  1398 = 'Time / Hour Angle'
  991 = 'Time during which the pressure is built up'
  992 = 'Time during which the pressure is built up [s]'
  993 = 'Time needed for stopping the pumps [s]'
  1347 = 'Time processing status (by C++ task)'
  753 = 'Time to wait after electronics power off [s]'
  701 = 'Time to wait after electronics power on [s]'
  729 = 'Time to wait after move [s]'
  702 = 'Time to wait before powering off automatically [s]'
  1338 = 'Time to wait while powering off the pumps [s]'
  1337 = 'Time to wait while powering on the pumps  [s]'
  1339 = 'Time to wait while powering on the pumps [s]'
  1045 = 'Timeout for a fast movement [s]'
  1044 = 'Timeout for a movement [s]'
  57 = 'Timeout when closing [s]'
  56 = 'Timeout when opening [s]'
  796 = 'Timer\n4 sec'
  797 = 'Timer\nOFF\ndelay\n4 sec'
  477 = 'Timestamp update toggle (heartbeat)'
  363 = 'Timestamps'
  794 = 'TOF'
  795 = 'TOF\n4 sec'
  2013 = 'Tolerance (in degrees) for AZI to determine if it is at a known position'
  2014 = 'Tolerance (in degrees) for ELE to determine if it is at a known position'
  2015 = 'Tolerance (in degrees) for ROC to determine if it is at a known position'
  2016 = 'Tolerance (in degrees) for RON to determine if it is at a known position'
  62 = 'Tolerance at closed position [°]'
  60 = 'Tolerance at open position [°]'
  61 = 'Tolerance for standing still [°/s]'
  1781 = 'TOO LOW'
  33 = 'TOP'
  426 = 'Top'
  709 = 'top'
  778 = 'TOP 1'
  783 = 'Top 1'
  933 = 'Top 1 no underpressure'
  851 = 'Top 1 underpressure'
  878 = 'Top 1 underpressure OK'
  779 = 'TOP 2'
  784 = 'Top 2'
  935 = 'Top 2 no underpressure'
  852 = 'Top 2 underpressure'
  879 = 'Top 2 underpressure OK'
  780 = 'TOP 3'
  786 = 'Top 3'
  936 = 'Top 3 no underpressure'
  853 = 'Top 3 underpressure'
  880 = 'Top 3 underpressure OK'
  781 = 'TOP 4'
  787 = 'Top 4'
  937 = 'Top 4 no underpressure'
  854 = 'Top 4 underpressure'
  881 = 'Top 4 underpressure OK'
  961 = 'TOP drive'
  942 = 'Top no overpressure'
  785 = 'Top OP 3'
  855 = 'Top overpressure'
  886 = 'Top overpressure OK'
  984 = 'Top setpoint:'
  890 = 'Top TRIP OK'
  2096 = 'Torque'
  1542 = 'Torque command'
  1216 = 'Total time in milliseconds to repeat the pattern'
  2062 = "TPoint azimuth (' A' ) sign (-1 is negative, 1 is positive)"
  2066 = "TPoint azimuth (' A' ) sign correction (-1 is negative, 1 is positive)"
  2064 = 'TPoint delta azimuth sign correction (-1 is negative, 1 is positive)'
  2067 = 'TPoint delta elevation sign correction (-1 is negative, 1 is positive)'
  2063 = "TPoint elevation ('E' ) sign (-1 is negative, 1 is positive)"
  2065 = "TPoint elevation ('E' ) sign correction (-1 is negative, 1 is positive)"
  2059 = 'TPoint invert azimuth (A)'
  2061 = "TPoint invert azimuth (input ' A' )"
  2060 = 'TPoint invert azimuth (input A)'
  2068 = 'TPoint: use old formulas (different sign convention)'
  1437 = 'Track target after pointing'
  1774 = 'Track the new target after pointing'
  1775 = 'Track the target'
  1435 = 'Tracking'
  1760 = 'Transformations status (by C++ task)'
  73 = 'TRANSLATION'
  330 = 'Translation'
  142 = 'Translation position [mm]'
  141 = 'Translation position [°]'
  270 = 'Translation status'
  407 = 'Transmission status'
  1979 = 'travelled'
  1367 = 'Tropospheric lapse rate [K/m]'
  1414 = 'Troubleshoot'
  1418 = 'Troubleshoot \n& restart'
  1419 = 'Troubleshoot \nand restart'
  1417 = 'Troubleshoot & restart'
  1415 = 'Troubleshooting\n& restarting'
  1420 = 'Troubleshooting \nand restarting'
  1712 = 'True if a positive torque must be applied, false if a negative torque must be applied'
  1715 = 'True if the ABL torque must be applied in the same direction as the AZI acceleration'
  1716 = 'True if the AZI and ABL axes rotate in the same direction'
  1713 = 'True if the AZI and ABL axes rotate in the same direction, false if NOT'
  1714 = 'True if the AZI and ABL axes rotate in the same direction, false if not'
  2102 = 'True position'
  1826 = 'TRUE to invert the counting direction of the absolute encoder'
  1827 = 'TRUE to invert the counting direction of the LIDAs'
  1100 = 'Tube accelerometers'
  1465 = 'Tube flexure - sin(zeta) law'
  1467 = 'Tube flexure - tan(zeta) law'
  1281 = 'Turn off Cassegrain derotator'
  1279 = 'Turn off Nasmyth B derotator'
  1280 = 'Turn on Cassegrain derotator'
  1278 = 'Turn on Nasmyth B derotator'
  1029 = 'Turn on/off the circulation pump manually'
  1333 = 'Turn on/off the pumps manually'
  1466 = 'TX'
  296 = 'TxError counter:'
  1128 = 'Unblock'
  1133 = 'Unblock\n(Only staff can unblock from GUI)'
  1127 = 'Unblock\n(STAFF)'
  1134 = 'Unblock\n(Unblock from GUI = STAFF ONLY)'
  1135 = 'Unblock\n(Unblock from GUI = staff only)'
  1131 = 'Unblock\nforever'
  1132 = 'Unblock\nuntil re-initialize'
  1136 = 'Unblock \npermanently\n(until re-initialization)'
  1202 = 'Unblock button is being pushed'
  1137 = 'Unblock permanently\n(until re-initialization)'
  1140 = 'Unblock permanently\n(until safety is re-initialialized)'
  1141 = 'Unblock permanently\n(until Safety is re-initialized)'
  1126 = 'Unblock telescope'
  1139 = 'Unblocked permanently'
  817 = 'Under\npressure'
  772 = 'Underpressure'
  950 = 'Underpressure error'
  951 = 'Underpressure error detection'
  877 = 'Underpressure OK'
  777 = 'Underpressure status'
  776 = 'Underpressure summary'
  770 = 'Underpressure top 1'
  771 = 'Underpressure top 2'
  1442 = 'Units'
  413 = 'Unlock'
  1541 = 'UNLOCK'
  1805 = 'Unlock brake'
  1809 = 'Unlock brake temporarily'
  1535 = 'Update the (non-cyclic) values below'
  1534 = 'Update the non-cyclic values below'
  1505 = 'Update the values below'
  1331 = 'Use Cassegrain derotator'
  1332 = 'Use Nasmyth B derotator'
  1361 = 'Use relative humidity from sensors (not the value below)'
  1364 = 'Use relative humidity from telemetry (not the value below)'
  1358 = 'Use temperature from sensors (not the value below)'
  1363 = 'Use temperature from telemetry (not the value below)'
  1355 = 'Use temperatures from sensors (not from config)'
  1356 = 'Use temperatures from sensors (not the value below)'
  1610 = 'UT1'
  369 = 'UTC'
  372 = 'UTC date (y-m-s)'
  373 = 'UTC date (y-m-s) :'
  375 = 'UTC date (year-month-day) :'
  384 = 'UTC date (years - months - days)'
  381 = 'UTC date (years - months - days) :'
  380 = 'UTC date (years-months-days) :'
  374 = 'UTC date (yyyy-mm-dd) :'
  383 = 'UTC time (hours : minutes : seconds)'
  382 = 'UTC time (hours : minutes : seconds) :'
  376 = 'UTC time (hours:minutes:seconds) :'
  371 = 'UTC year/month/day'
  370 = 'UTC:'
  617 = 'Vacuum'
  618 = 'Vacuum OFF'
  643 = 'Vacuum ON'
  646 = 'Vacuum relay'
  173 = 'Value to write'
  120 = 'Vel. control Prop. term'
  122 = 'Vel. ctrl. Integral term'
  121 = 'Vel. ctrl. Proport. term'
  1738 = 'Velocities'
  1838 = 'Velocity'
  1683 = 'Velocity limit (bidirectional) of the physical axis in degrees/sec (>0)'
  1682 = 'Velocity limit (both directions) of the physical axis in degrees/sec (>0)'
  1679 = 'Velocity limit of the physical axis in degrees/sec (>0)'
  1720 = 'Velocity to search for the homing mark, in degrees/sec'
  1719 = 'Velocity when going to the start position, in degrees/sec'
  1292 = 'Verify fixed positions on thermal focus'
  836 = 'Verify if '
  837 = 'Verify if \nfrequency'
  838 = 'Verify if \nfrequency rises'
  839 = 'Verify if pumps\nfrequency rises'
  840 = 'Verify if pumps\nfrequency rises\n(QMin -> 0)'
  1463 = 'Vertical displacement of Nasmyth rotator'
  1621 = 'Virtual axis'
  1565 = 'W 270°'
  964 = 'Wait 2 minutes, so that the system can full start up in the background.'
  972 = 'Wait 2 minutes, so that the system can fully start up in the background.'
  1411 = 'Wake up'
  1427 = 'Wake up ...'
  1409 = 'Wake up telescope'
  1423 = 'Wake up the telescope'
  7 = 'WcState:'
  1657 = 'Which input (0-7) represents the negative limit switch?'
  1656 = 'Which input (0-7) represents the positive limit switch?'
  579 = 'with: RadialPressureSetpoint = CorrectionCoefficient * 1.33 bar * cos(elevation)'
  172 = 'Write'
  176 = 'Write config at initialization'
  688 = 'X'
  1106 = 'X angle'
  1285 = 'X fixed position tolerance [mm]'
  1284 = 'X fixed position [mm]'
  1 = 'XML config'
  150 = 'XML file'
  689 = 'Y'
  1287 = 'Y fixed position tolerance [mm]'
  1286 = 'Y fixed position [mm]'
  686 = 'Z'
  1077 = 'Z axis:'
  1255 = 'Z high speed'
  21 = '°'
  22 = '°/s'
  1758 = 'α'
  1856 = 'α offsetted'
  1854 = 'α travelled'
  1759 = 'δ'
  1858 = 'δ offsetted'
  1857 = 'δ travelled'
END_TEXTLIST

// ---- MTCS/Axes/Visu/VISU_AxesAzimuthAxis.TcVIS
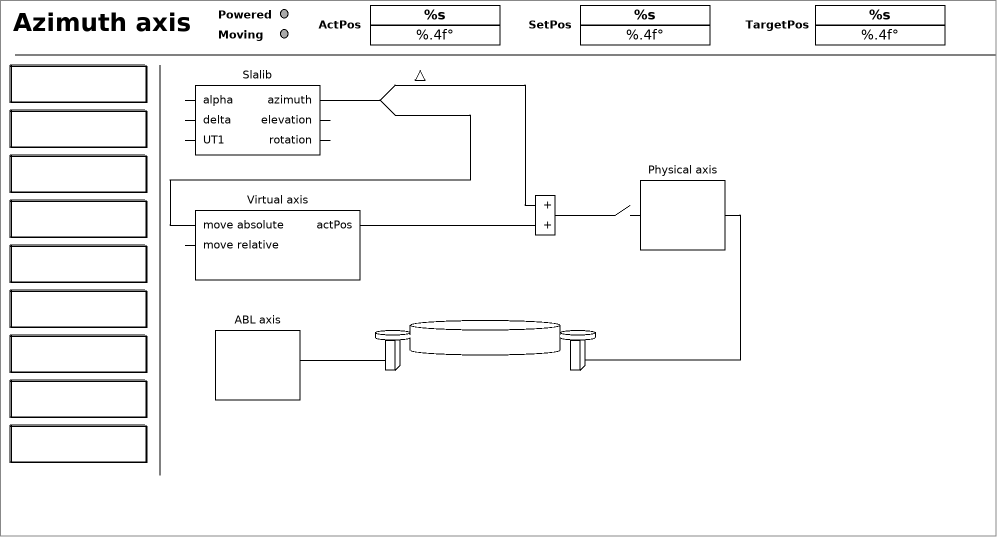
VISUALIZATION VISU_AxesAzimuthAxis  // 997x537
VAR_IN_OUT
	ref : AxesAzimuthAxis;
    ref_aziDriveChannel : AX52XXDriveChannel;
    ref_ablDriveChannel : AX52XXDriveChannel;
    widget : AxesAzimuthAxisWidget;
END_VAR
    Rectangle (10,0 195x45), "Azimuth axis"
    Frame (10,65 140x40)
        shows VISU_SubSubSystemButton(widget := widget.button_overview)
        OnMouseClick: FrameSelectionChange Selection=SelectedFrame=26eb0533-0645-4710-820d-78aa3cb40b18, GlobSel=AssignType=Directly, SelType=Locally
        OnMouseClick: execute { widget.activeTab := AxesAzimuthAxisTabs.OVERVIEW; }
    Frame (165,65 805x470)
        shows VISU_AxesAzimuthAxis_Overview(ref := ref, widget := widget)
        shows VISU_AxesAzimuthAxis_Processes(ref := ref, ref_aziDriveChannel := ref_aziDriveChannel, widget := widget)
        shows VISU_AX522DriveChannel(ref := ref_aziDriveChannel, widget := widget.aziDriveChannel)
        shows VISU_AX522DriveChannel(ref := ref_ablDriveChannel, widget := widget.ablDriveChannel)
        shows VISU_AngularAxis(axis := ref.parts.virtualAxis, widget := widget.virtualAxis)
        shows VISU_AngularAxis(axis := ref.parts.physicalAxis, widget := widget.physicalAxis)
        shows VISU_AngularAxis(axis := ref.parts.ablAxis, widget := widget.ablAxis)
        shows VISU_AxesAzimuthAxis_Lidas(ref := ref, widget := widget)
        shows VISU_AxesAzimuthAxis_AbsoluteEncoder(ref := ref, widget := widget)
        p4174417010: ref.parts.virtualAxis
        p2620823199: ref
    Line (160,475) (160,65)
    Frame (10,155 140x40)
        shows VISU_SubSubSystemButton(widget := widget.button_aziDriveChannel)
        OnMouseClick: FrameSelectionChange Selection=SelectedFrame=26eb0533-0645-4710-820d-78aa3cb40b18, Selection=2, GlobSel=AssignType=Directly, SelType=Locally
        OnMouseClick: execute { widget.activeTab := AxesAzimuthAxisTabs.AZI_DRIVE_CHANNEL; }
    Frame (10,200 140x40)
        shows VISU_SubSubSystemButton(widget := widget.button_ablDriveChannel)
        OnMouseClick: FrameSelectionChange Selection=SelectedFrame=26eb0533-0645-4710-820d-78aa3cb40b18, Selection=3, GlobSel=AssignType=Directly, SelType=Locally
        OnMouseClick: execute { widget.activeTab := AxesAzimuthAxisTabs.ABL_DRIVE_CHANNEL; }
    Frame (10,245 140x40)
        shows VISU_SubSubSystemButton(widget := widget.button_virtualAxis)
        OnMouseClick: FrameSelectionChange Selection=SelectedFrame=26eb0533-0645-4710-820d-78aa3cb40b18, Selection=4, GlobSel=AssignType=Directly, SelType=Locally
        OnMouseClick: execute { widget.activeTab := AxesAzimuthAxisTabs.VIRTUAL_AXIS; }
    Frame (10,290 140x40)
        shows VISU_SubSubSystemButton(widget := widget.button_physicalAxis)
        OnMouseClick: FrameSelectionChange Selection=SelectedFrame=26eb0533-0645-4710-820d-78aa3cb40b18, Selection=5, GlobSel=AssignType=Directly, SelType=Locally
        OnMouseClick: execute { widget.activeTab := AxesAzimuthAxisTabs.PHYSICAL_AXIS; }
    Frame (10,335 140x40)
        shows VISU_SubSubSystemButton(widget := widget.button_ablAxis)
        OnMouseClick: FrameSelectionChange Selection=SelectedFrame=26eb0533-0645-4710-820d-78aa3cb40b18, Selection=6, GlobSel=AssignType=Directly, SelType=Locally
        OnMouseClick: execute { widget.activeTab := AxesAzimuthAxisTabs.ABL_AXIS; }
    Frame (10,380 140x40)
        shows VISU_SubSubSystemButton(widget := widget.button_lidas)
        OnMouseClick: FrameSelectionChange Selection=SelectedFrame=26eb0533-0645-4710-820d-78aa3cb40b18, Selection=7, GlobSel=AssignType=Directly, SelType=Locally
        OnMouseClick: execute { widget.activeTab := AxesAzimuthAxisTabs.LIDAS; }
    Frame (10,425 140x40)
        shows VISU_SubSubSystemButton(widget := widget.button_absoluteEncoder)
        OnMouseClick: FrameSelectionChange Selection=SelectedFrame=26eb0533-0645-4710-820d-78aa3cb40b18, Selection=8, GlobSel=AssignType=Directly, SelType=Locally
        OnMouseClick: execute { widget.activeTab := AxesAzimuthAxisTabs.ABSOLUTE_ENCODER; }
    Frame (10,110 140x40)
        shows VISU_SubSubSystemButton(widget := widget.button_processes)
        OnMouseClick: FrameSelectionChange Selection=SelectedFrame=26eb0533-0645-4710-820d-78aa3cb40b18, Selection=1, GlobSel=AssignType=Directly, SelType=Locally
        OnMouseClick: execute { widget.activeTab := AxesAzimuthAxisTabs.PROCESSES; }
    Line (995,55) (15,55)
    Label (310,0 60x50), "ActPos"
    Rectangle (370,5 130x20), "%s", text variable: widget.actPos.dmsString
    Rectangle (370,25 130x20), "%.4f°", text variable: ref.actPos.degrees.value
    Label (520,0 60x50), "SetPos"
    Rectangle (580,5 130x20), "%s", text variable: widget.setPos.dmsString
    Rectangle (580,25 130x20), "%.4f°", text variable: ref.setPos.degrees.value
    Label (740,0 75x50), "TargetPos"
    Rectangle (815,5 130x20), "%s", text variable: widget.targetPos.dmsString
    Rectangle (815,25 130x20), "%.4f°", text variable: ref.targetPos.degrees.value
    Label (215,5 65x20), "Powered"
    Frame (280,5 10x15)
        shows VISU_State_gray_green(state := ref.statuses.poweredStatus.enabled)
    Label (215,25 65x20), "Moving"
    Frame (280,25 10x15)
        shows VISU_State_gray_green(state := ref.parts.physicalAxis.axis_ref.Status.Moving)
END_VISUALIZATION

// ---- MTCS/Axes/Visu/VISU_AxesAzimuthAxis_AbsoluteEncoder.TcVIS
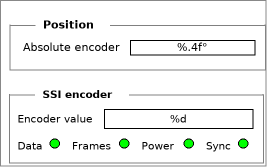
VISUALIZATION VISU_AxesAzimuthAxis_AbsoluteEncoder  // 267x167
VAR_IN_OUT
	ref : AxesAzimuthAxis;
    widget : AxesAzimuthAxisWidget;
END_VAR
    Frame (-5,80 270x85)
        shows VISU_SSIEncoder(ref := ref.parts.absoluteEncoder)
    Label (40,15 65x20), "Position"
    Polyline (110,25) (265,25) (265,70) (10,70) (10,25) (35,25)
    Label (20,40 105x15), "Absolute encoder"
    Rectangle (130,40 125x15), "%.4f°", text variable: ref.absoluteEncoderPosition.degrees.value
END_VISUALIZATION

// ---- MTCS/Axes/Visu/VISU_AxesAzimuthAxis_Processes.TcVIS
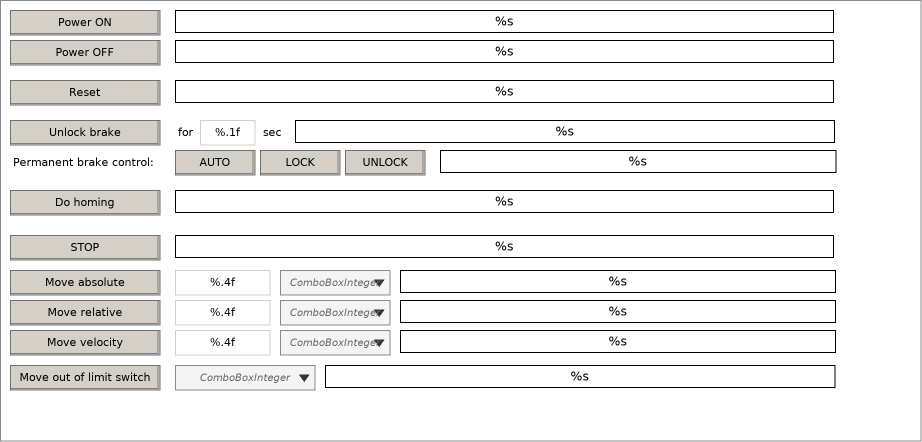
VISUALIZATION VISU_AxesAzimuthAxis_Processes  // 922x442
VAR_IN_OUT
	ref : AxesAzimuthAxis;
    ref_aziDriveChannel : AX52XXDriveChannel;
    widget : AxesAzimuthAxisWidget;
END_VAR
    Frame (10,10 910x55)
        shows VISU_Axes_Commands_Power(powerOn := ref.processes.powerOn, powerOff := ref.processes.powerOff, powerOnStatus := widget.processes_powerOnStatus, powerOffStatus := widget.processes_powerOffStatus)
    Frame (10,80 910x25)
        shows VISU_Axes_Commands_Reset(reset := ref.processes.reset, resetStatus := widget.processes_resetStatus)
    Frame (10,120 910x55)
        shows VISU_Axes_Commands_Brake(unlockBrake := ref.processes.unlockBrake, setBrake := ref_aziDriveChannel.processes.setBrake, unlockBrakeStatus := widget.processes_unlockBrakeStatus, setBrakeStatus := widget.aziDriveChannel.processes_setBrakeStatus)
    Frame (10,190 910x35)
        shows VISU_Axes_Commands_DoHoming(doHoming := ref.processes.doHoming, doHomingStatus := widget.processes_doHomingStatus)
    Frame (10,235 910x205)
        shows VISU_Axes_Commands_Movement(stop := ref.processes.stop, moveOutOfLimitSwitch := ref.processes.moveOutOfLimitSwitch, moveAbsolute := ref.processes.moveAbsolute, moveRelative := ref.processes.moveRelative, moveVelocity := ref.processes.moveVelocity, stopStatus := widget.processes_stopStatus, moveOutOfLimitSwitchStatus := widget.processes_moveOutOfLimitSwitchStatus, moveAbsoluteStatus := widget.processes_moveAbsoluteStatus, moveRelativeStatus := widget.processes_moveRelativeStatus, moveVelocityStatus := widget.processes_moveVelocityStatus)
END_VISUALIZATION

// ---- MTCS/Axes/Visu/VISU_AxesConfig_KnownPosition.TcVIS
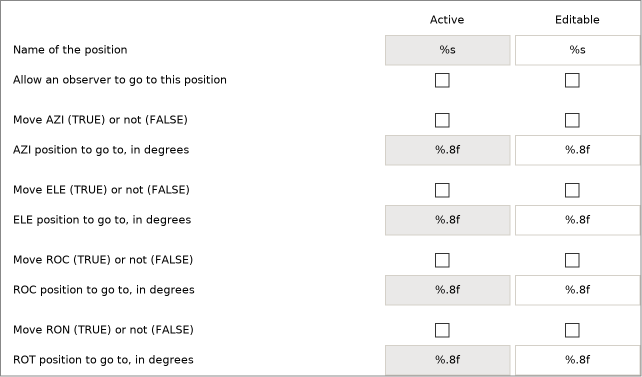
VISUALIZATION VISU_AxesConfig_KnownPosition  // 642x377
VAR_IN_OUT
    editable : AxesKnownPositionConfig;
	active : AxesKnownPositionConfig;
END_VAR
    Frame (385,35 255x30)
        shows VISU_ConfigStringEntry(active := active.name, editable := editable.name)
    Label (385,10 125x20), "Active"
    Label (515,10 125x20), "Editable"
    Label (10,35 370x30), "Name of the position"
    Frame (385,65 255x30)
        shows VISU_ConfigBOOLEntry(active := active.allowObserver, editable := editable.allowObserver)
    Label (10,65 370x30), "Allow an observer to go to this position"
    Label (10,135 370x30), "AZI position to go to, in degrees"
    Frame (385,135 255x30)
        shows VISU_ConfigLREAL8Entry(active := active.azi, editable := editable.azi)
    Label (10,105 370x30), "Move AZI (TRUE) or not (FALSE)"
    Frame (385,105 255x30)
        shows VISU_ConfigBOOLEntry(active := active.doAzi, editable := editable.doAzi)
    Label (10,205 370x30), "ELE position to go to, in degrees"
    Frame (385,205 255x30)
        shows VISU_ConfigLREAL8Entry(active := active.ele, editable := editable.ele)
    Label (10,175 370x30), "Move ELE (TRUE) or not (FALSE)"
    Frame (385,175 255x30)
        shows VISU_ConfigBOOLEntry(active := active.doEle, editable := editable.doEle)
    Label (10,275 370x30), "ROC position to go to, in degrees"
    Frame (385,275 255x30)
        shows VISU_ConfigLREAL8Entry(active := active.roc, editable := editable.roc)
    Label (10,245 370x30), "Move ROC (TRUE) or not (FALSE)"
    Frame (385,245 255x30)
        shows VISU_ConfigBOOLEntry(active := active.doRoc, editable := editable.doRoc)
    Label (10,345 370x30), "ROT position to go to, in degrees"
    Frame (385,345 255x30)
        shows VISU_ConfigLREAL8Entry(active := active.ron, editable := editable.ron)
    Label (10,315 370x30), "Move RON (TRUE) or not (FALSE)"
    Frame (385,315 255x30)
        shows VISU_ConfigBOOLEntry(active := active.doRon, editable := editable.doRon)
END_VISUALIZATION

// ---- MTCS/Axes/Visu/VISU_AxesConfig_KnownPositions.TcVIS
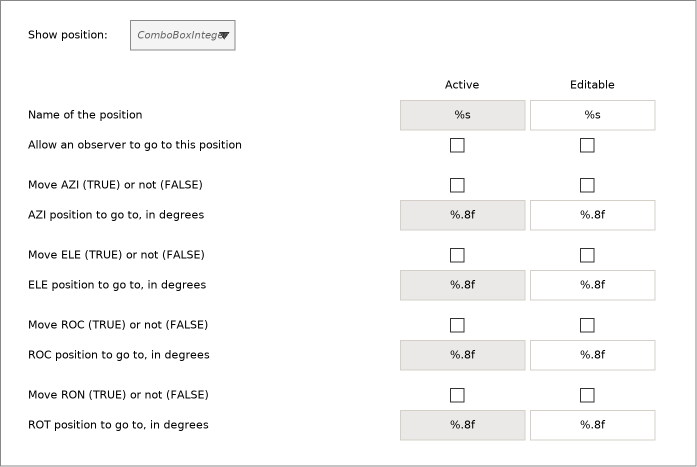
VISUALIZATION VISU_AxesConfig_KnownPositions  // 697x467
VAR_IN_OUT
    activePosition : INT;
    editable : AxesKnownPositionsConfig;
	active : AxesKnownPositionsConfig;
END_VAR
    Frame (15,65 680x400), frame switch variable: activePosition
        shows VISU_AxesConfig_KnownPosition(editable := editable.position0, active := active.position0)
        shows VISU_AxesConfig_KnownPosition(editable := editable.position1, active := active.position1)
        shows VISU_AxesConfig_KnownPosition(editable := editable.position2, active := active.position2)
        shows VISU_AxesConfig_KnownPosition(editable := editable.position3, active := active.position3)
        shows VISU_AxesConfig_KnownPosition(editable := editable.position4, active := active.position4)
        shows VISU_AxesConfig_KnownPosition(editable := editable.position5, active := active.position5)
        shows VISU_AxesConfig_KnownPosition(editable := editable.position6, active := active.position6)
        shows VISU_AxesConfig_KnownPosition(editable := editable.position7, active := active.position7)
        shows VISU_AxesConfig_KnownPosition(editable := editable.position8, active := active.position8)
        shows VISU_AxesConfig_KnownPosition(editable := editable.position9, active := active.position9)
        shows VISU_AxesConfig_KnownPosition(editable := editable.position10, active := active.position10)
        shows VISU_AxesConfig_KnownPosition(editable := editable.position11, active := active.position11)
        shows VISU_AxesConfig_KnownPosition(editable := editable.position12, active := active.position12)
        shows VISU_AxesConfig_KnownPosition(editable := editable.position13, active := active.position13)
        shows VISU_AxesConfig_KnownPosition(editable := editable.position14, active := active.position14)
        shows VISU_AxesConfig_KnownPosition(editable := editable.position15, active := active.position15)
        shows VISU_AxesConfig_KnownPosition(editable := editable.position16, active := active.position16)
        shows VISU_AxesConfig_KnownPosition(editable := editable.position17, active := active.position17)
        shows VISU_AxesConfig_KnownPosition(editable := editable.position18, active := active.position18)
        shows VISU_AxesConfig_KnownPosition(editable := editable.position19, active := active.position19)
    Label (25,20 150x30), "Show position:"
    ComboBoxInteger (130,20 105x30), variable: activePosition
END_VISUALIZATION

// ---- MTCS/Axes/Visu/VISU_AxesImage.TcVIS
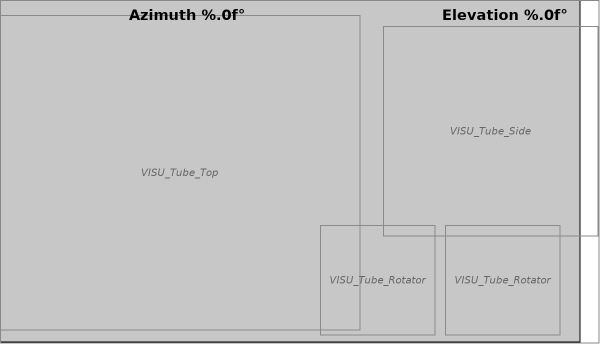
VISUALIZATION VISU_AxesImage  // 600x344
VAR_IN_OUT
	ref : Axes;
    widget : AxesWidget;
END_VAR
    Rectangle (0,0 580x342)
    Frame (383,26 215x210)
        shows VISU_Tube_Side(ele := widget.image.ele, eleTarget := widget.image.eleTarget, eleTargetInvisible := widget.image.eleTargetInvisible, mark10Degrees := widget.image.mark10Degrees)
    Frame (0,15 360x315)
        shows VISU_Tube_Top(widget := widget.image)
    Rectangle (90,5 195x20), "Azimuth %.0f°", text variable: ref.feedback.aziPos.degrees.value
    Rectangle (435,5 140x20), "Elevation %.0f°", text variable: ref.feedback.elePos.degrees.value
    Frame (320,225 115x110)
        shows VISU_Tube_Rotator(stationName := widget.image.rocStationName, name := widget.image.rocName, rotAngle := widget.image.roc)
    Frame (445,225 115x110)
        shows VISU_Tube_Rotator(stationName := widget.image.ronStationName, name := widget.image.ronName, rotAngle := widget.image.ron)
END_VISUALIZATION

// ---- MTCS/Axes/Visu/VISU_AxesManual_Offsets_AlphaDeltaRot.TcVIS
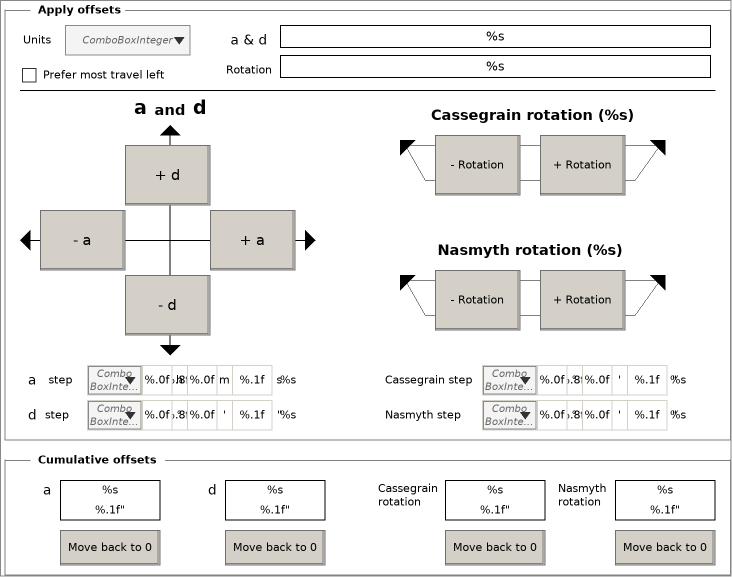
VISUALIZATION VISU_AxesManual_Offsets_AlphaDeltaRot  // 732x577
VAR_IN_OUT
	ref : Axes;
    widget : AxesManualOffsetsWidget;
END_VAR
    Polyline (165,460) (730,460) (730,575) (5,575) (5,460) (30,460)
    Polyline (125,10) (730,10) (730,440) (5,440) (5,10) (30,10)
    Polygon (660,145) (635,180) (425,180) (405,145)
    Line (170,350) (170,130)
    Line (25,240) (315,240)
    ComboBoxInteger (65,25 125x30), variable: widget.moveRelative.units, text list: 'AxesMoveAlphaDeltaProcessUnitsTextList'
    Rectangle (277,365 35x30), "%s", text variable: widget.pointRelative.unitsText, invisible if: widget.pointRelative.units = AxesMoveProcessWidgetUnits.DEGMINSEC
    Textfield (87,365 180x30), "%.8f", text variable: widget.pointRelative.field_alpha_decimal, invisible if: widget.pointRelative.units = AxesMoveProcessWidgetUnits.DEGMINSEC, input disabled if: widget.pointRelative.alphaDisabled
        OnMouseClick: write the text variable via VisuDialogs.Numpad
    Textfield (142,365 30x30), "%.0f", text variable: widget.pointRelative.field_alpha_h, invisible if: widget.pointRelative.units <> AxesMoveProcessWidgetUnits.DEGMINSEC, input disabled if: widget.pointRelative.alphaDisabled
        OnMouseClick: write the text variable via VisuDialogs.Numpad
    ComboBoxInteger (88,366 53x28), variable: widget.pointRelative.field_alpha_sign, invisible if: widget.pointRelative.units <> AxesMoveProcessWidgetUnits.DEGMINSEC, input disabled if: widget.pointRelative.alphaDisabled, text list: 'AxesDialogSignTextList'
    Textfield (187,365 30x30), "%.0f", text variable: widget.pointRelative.field_alpha_m, invisible if: widget.pointRelative.units <> AxesMoveProcessWidgetUnits.DEGMINSEC, input disabled if: widget.pointRelative.alphaDisabled
        OnMouseClick: write the text variable via VisuDialogs.Numpad
    Textfield (232,365 40x30), "%.1f", text variable: widget.pointRelative.field_alpha_s, invisible if: widget.pointRelative.units <> AxesMoveProcessWidgetUnits.DEGMINSEC, input disabled if: widget.pointRelative.alphaDisabled
        OnMouseClick: write the text variable via VisuDialogs.Numpad
    Label (172,365 15x30), "h", invisible if: widget.moveRelative.units <> AxesMoveProcessWidgetUnits.DEGMINSEC
    Label (217,365 15x30), "m", invisible if: widget.pointRelative.units <> AxesMoveProcessWidgetUnits.DEGMINSEC
    Label (272,365 15x30), "s", invisible if: widget.pointRelative.units <> AxesMoveProcessWidgetUnits.DEGMINSEC
    Rectangle (277,400 35x30), "%s", text variable: widget.pointRelative.unitsText, invisible if: widget.pointRelative.units = AxesMoveProcessWidgetUnits.DEGMINSEC
    Textfield (87,400 180x30), "%.8f", text variable: widget.pointRelative.field_delta_decimal, invisible if: widget.pointRelative.units = AxesMoveProcessWidgetUnits.DEGMINSEC, input disabled if: widget.pointRelative.deltaDisabled
        OnMouseClick: write the text variable via VisuDialogs.Numpad
    Textfield (142,400 30x30), "%.0f", text variable: widget.pointRelative.field_delta_d, invisible if: widget.pointRelative.units <> AxesMoveProcessWidgetUnits.DEGMINSEC, input disabled if: widget.pointRelative.deltaDisabled
        OnMouseClick: write the text variable via VisuDialogs.Numpad
    ComboBoxInteger (88,401 53x28), variable: widget.pointRelative.field_delta_sign, invisible if: widget.pointRelative.units <> AxesMoveProcessWidgetUnits.DEGMINSEC, input disabled if: widget.pointRelative.deltaDisabled, text list: 'AxesDialogSignTextList'
    Textfield (187,400 30x30), "%.0f", text variable: widget.pointRelative.field_delta_m, invisible if: widget.pointRelative.units <> AxesMoveProcessWidgetUnits.DEGMINSEC, input disabled if: widget.pointRelative.deltaDisabled
        OnMouseClick: write the text variable via VisuDialogs.Numpad
    Textfield (232,400 40x30), "%.1f", text variable: widget.pointRelative.field_delta_s, invisible if: widget.pointRelative.units <> AxesMoveProcessWidgetUnits.DEGMINSEC, input disabled if: widget.pointRelative.deltaDisabled
        OnMouseClick: write the text variable via VisuDialogs.Numpad
    Label (172,400 15x30), "°", invisible if: widget.moveRelative.units <> AxesMoveProcessWidgetUnits.DEGMINSEC
    Label (217,400 15x30), "'", invisible if: widget.moveRelative.units <> AxesMoveProcessWidgetUnits.DEGMINSEC
    Label (272,400 15x30), """, invisible if: widget.pointRelative.units <> AxesMoveProcessWidgetUnits.DEGMINSEC
    Rectangle (667,365 35x30), "%s", text variable: widget.moveRelative.unitsText, invisible if: widget.moveRelative.units = AxesMoveProcessWidgetUnits.DEGMINSEC
    Textfield (482,365 180x30), "%.8f", text variable: widget.moveRelative.field_roc_decimal, invisible if: widget.moveRelative.units = AxesMoveProcessWidgetUnits.DEGMINSEC, input disabled if: widget.moveRelative.rocDisabled
        OnMouseClick: write the text variable via VisuDialogs.Numpad
    Textfield (537,365 30x30), "%.0f", text variable: widget.moveRelative.field_roc_d, invisible if: widget.moveRelative.units <> AxesMoveProcessWidgetUnits.DEGMINSEC, input disabled if: widget.moveRelative.rocDisabled
        OnMouseClick: write the text variable via VisuDialogs.Numpad
    ComboBoxInteger (483,366 53x28), variable: widget.moveRelative.field_roc_sign, invisible if: widget.moveRelative.units <> AxesMoveProcessWidgetUnits.DEGMINSEC, input disabled if: widget.moveRelative.rocDisabled, text list: 'AxesDialogSignTextList'
    Textfield (582,365 30x30), "%.0f", text variable: widget.moveRelative.field_roc_m, invisible if: widget.moveRelative.units <> AxesMoveProcessWidgetUnits.DEGMINSEC, input disabled if: widget.moveRelative.rocDisabled
        OnMouseClick: write the text variable via VisuDialogs.Numpad
    Textfield (627,365 40x30), "%.1f", text variable: widget.moveRelative.field_roc_s, invisible if: widget.moveRelative.units <> AxesMoveProcessWidgetUnits.DEGMINSEC, input disabled if: widget.moveRelative.rocDisabled
        OnMouseClick: write the text variable via VisuDialogs.Numpad
    Label (567,365 15x30), "°", invisible if: widget.moveRelative.units <> AxesMoveProcessWidgetUnits.DEGMINSEC
    Label (612,365 15x30), "'", invisible if: widget.moveRelative.units <> AxesMoveProcessWidgetUnits.DEGMINSEC
    Label (667,365 15x30), """, invisible if: widget.moveRelative.units <> AxesMoveProcessWidgetUnits.DEGMINSEC
    Rectangle (667,400 35x30), "%s", text variable: widget.moveRelative.unitsText, invisible if: widget.moveRelative.units = AxesMoveProcessWidgetUnits.DEGMINSEC
    Textfield (482,400 180x30), "%.8f", text variable: widget.moveRelative.field_ron_decimal, invisible if: widget.moveRelative.units = AxesMoveProcessWidgetUnits.DEGMINSEC, input disabled if: widget.moveRelative.ronDisabled
        OnMouseClick: write the text variable via VisuDialogs.Numpad
    Textfield (537,400 30x30), "%.0f", text variable: widget.moveRelative.field_ron_d, invisible if: widget.moveRelative.units <> AxesMoveProcessWidgetUnits.DEGMINSEC, input disabled if: widget.moveRelative.ronDisabled
        OnMouseClick: write the text variable via VisuDialogs.Numpad
    ComboBoxInteger (483,401 53x28), variable: widget.moveRelative.field_ron_sign, invisible if: widget.moveRelative.units <> AxesMoveProcessWidgetUnits.DEGMINSEC, input disabled if: widget.moveRelative.ronDisabled, text list: 'AxesDialogSignTextList'
    Textfield (582,400 30x30), "%.0f", text variable: widget.moveRelative.field_ron_m, invisible if: widget.moveRelative.units <> AxesMoveProcessWidgetUnits.DEGMINSEC, input disabled if: widget.moveRelative.ronDisabled
        OnMouseClick: write the text variable via VisuDialogs.Numpad
    Textfield (627,400 40x30), "%.1f", text variable: widget.moveRelative.field_ron_s, invisible if: widget.moveRelative.units <> AxesMoveProcessWidgetUnits.DEGMINSEC, input disabled if: widget.moveRelative.ronDisabled
        OnMouseClick: write the text variable via VisuDialogs.Numpad
    Label (567,400 15x30), "°", invisible if: widget.moveRelative.units <> AxesMoveProcessWidgetUnits.DEGMINSEC
    Label (612,400 15x30), "'", invisible if: widget.moveRelative.units <> AxesMoveProcessWidgetUnits.DEGMINSEC
    Label (667,400 15x30), """, invisible if: widget.moveRelative.units <> AxesMoveProcessWidgetUnits.DEGMINSEC
    Frame (280,25 435x25)
        shows VISU_StatusWidget(widget := widget.pointRelative.actualStatus)
    Label (35,0 100x20), "Apply offsets"
    Button (125,145 85x60), "+ d", input disabled if: widget.pointRelative.deltaDisabled
        OnMouseClick: execute {
            ref.processes.pointRelative.request(
                alphaUnits := AxesAlphaUnits.DEGREES,
                alpha := 0.0,
                deltaunits := AxesDeltaUnits.DEGREES,
                delta := widget.pointRelative.deltaDeg);
        }
    Button (125,275 85x60), "- d", input disabled if: widget.pointRelative.deltaDisabled
        OnMouseClick: execute {
            ref.processes.pointRelative.request(
                alphaUnits := AxesAlphaUnits.DEGREES,
                alpha := 0.0,
                deltaunits := AxesDeltaUnits.DEGREES,
                delta := -widget.pointRelative.deltaDeg);
        }
    Button (210,210 85x60), "+ a", input disabled if: widget.pointRelative.alphaDisabled
        OnMouseClick: execute {
            ref.processes.pointRelative.request(
                alphaUnits := AxesAlphaUnits.DEGREES,
                alpha := widget.pointRelative.alphaDeg,
                deltaunits := AxesDeltaUnits.DEGREES,
                delta := 0.0);
        }
    Button (40,210 85x60), "- a", input disabled if: widget.pointRelative.alphaDisabled
        OnMouseClick: execute {
            ref.processes.pointRelative.request(
                alphaUnits := AxesAlphaUnits.DEGREES,
                alpha := -widget.pointRelative.alphaDeg,
                deltaunits := AxesDeltaUnits.DEGREES,
                delta := 0.0);
        }
    Label (42,365 35x30), "step"
    Label (42,400 40x30), "step"
    Button (540,135 85x60), "+ Rotation", input disabled if: widget.moveRelative.rocDisabled
        OnMouseClick: execute {
            ref.processes.moveRelative.request(
                units := AxesMoveUnits.DEGREES,
                azi := 0.0,
                ele := 0.0,
                rot := 0.0,
                roc := widget.moveRelative.rocDeg,
                ron := 0.0,
                doAzi := FALSE,
                doEle := FALSE,
                doRot := FALSE,
                doRoc := TRUE,
                doRon := FALSE,
                preferMostTravel := widget.preferMostTravel);
        }
    Button (435,135 85x60), "- Rotation", input disabled if: widget.moveRelative.rocDisabled
        OnMouseClick: execute {
            ref.processes.moveRelative.request(
                units := AxesMoveUnits.DEGREES,
                azi := 0.0,
                ele := 0.0,
                rot := 0.0,
                roc := -widget.moveRelative.rocDeg,
                ron := 0.0,
                doAzi := FALSE,
                doEle := FALSE,
                doRot := FALSE,
                doRoc := TRUE,
                doRon := FALSE,
                preferMostTravel := widget.preferMostTravel);
        }
    Polygon (160,135) (170,125) (180,135)
    Polygon (30,250) (20,240) (30,230)
    Polygon (305,250) (315,240) (305,230)
    Polygon (160,345) (170,355) (180,345)
    Polygon (665,155) (665,140) (650,140)
    Polygon (400,155) (415,140) (400,140)
    Label (382,365 100x30), "Cassegrain step"
    Label (382,400 100x30), "Nasmyth step"
    Label (20,25 55x30), "Units"
    Label (220,25 50x30), "a & d"
    Line (20,90) (715,90)
    Polygon (660,280) (635,315) (425,315) (405,280)
    Button (540,270 85x60), "+ Rotation", input disabled if: widget.moveRelative.ronDisabled
        OnMouseClick: execute {
            ref.processes.moveRelative.request(
                units := AxesMoveUnits.DEGREES,
                azi := 0.0,
                ele := 0.0,
                rot := 0.0,
                roc := 0.0,
                ron := widget.moveRelative.ronDeg,
                doAzi := FALSE,
                doEle := FALSE,
                doRot := FALSE,
                doRoc := FALSE,
                doRon := TRUE,
                preferMostTravel := widget.preferMostTravel);
        }
    Button (435,270 85x60), "- Rotation", input disabled if: widget.moveRelative.ronDisabled
        OnMouseClick: execute {
            ref.processes.moveRelative.request(
                units := AxesMoveUnits.DEGREES,
                azi := 0.0,
                ele := 0.0,
                rot := 0.0,
                roc := 0.0,
                ron := -widget.moveRelative.ronDeg,
                doAzi := FALSE,
                doEle := FALSE,
                doRot := FALSE,
                doRoc := FALSE,
                doRon := TRUE,
                preferMostTravel := widget.preferMostTravel);
        }
    Polygon (665,290) (665,275) (650,275)
    Polygon (400,290) (415,275) (400,275)
    Label (145,95 50x30), "and"
    Label (25,400 20x30), "d"
    Label (25,365 20x30), "a"
    Label (190,90 40x35), "d"
    Label (110,90 40x35), "a"
    Label (205,55 70x30), "Rotation"
    Frame (280,55 435x25)
        shows VISU_StatusWidget(widget := widget.moveRelative.actualStatus)
    Rectangle (60,480 100x20), "%s", text variable: widget.alphaOffsetted.hmsString
    Label (40,475 20x30), "a"
    Rectangle (60,500 100x20), "%.1f"", text variable: ref.target.alphaOffsetted.arcseconds.value
    Label (205,475 20x30), "d"
    Button (60,530 100x35), "Move back to 0", input disabled if: widget.pointRelative.alphaDisabled
        OnMouseClick: execute {
            ref.processes.pointRelative.request(
                alphaUnits := AxesAlphaUnits.DEGREES,
                alpha := -ref.target.alphaOffsetted.degrees.value,
                deltaunits := AxesDeltaUnits.DEGREES,
                delta := 0.0);
        }
    Label (35,450 120x20), "Cumulative offsets"
    Rectangle (60,480 100x40), colour toggle: widget.pointRelative.alphaDisabled
    Rectangle (225,480 100x20), "%s", text variable: widget.deltaOffsetted.dmsString
    Rectangle (225,500 100x20), "%.1f"", text variable: ref.target.deltaOffsetted.arcseconds.value
    Button (225,530 100x35), "Move back to 0", input disabled if: widget.pointRelative.deltaDisabled
        OnMouseClick: execute {
            ref.processes.pointRelative.request(
                alphaUnits := AxesAlphaUnits.DEGREES,
                alpha := 0.0,
                deltaunits := AxesDeltaUnits.DEGREES,
                delta := -ref.target.deltaOffsetted.degrees.value);
        }
    Rectangle (225,480 100x40), colour toggle: widget.pointRelative.deltaDisabled
    Rectangle (445,480 100x20), "%s", text variable: widget.rocTargetOffset.dmsString
    Rectangle (445,500 100x20), "%.1f"", text variable: ref.parts.roc.targetOffset.arcseconds.value
    Button (445,530 100x35), "Move back to 0", input disabled if: widget.moveRelative.rocDisabled
        OnMouseClick: execute {
            ref.processes.moveRelative.request(
                units := AxesMoveUnits.DEGREES,
                azi := 0.0,
                ele := 0.0,
                rot := 0.0,
                roc := -ref.parts.roc.targetOffset.degrees.value,
                ron := 0.0,
                doAzi := FALSE,
                doEle := FALSE,
                doRot := FALSE,
                doRoc := TRUE,
                doRon := FALSE, preferMostTravel := widget.preferMostTravel);
        }
    Rectangle (445,480 100x40), colour toggle: widget.moveRelative.rocDisabled
    Label (375,480 70x30), "Cassegrain rotation"
    Rectangle (615,480 100x20), "%s", text variable: widget.ronTargetOffset.dmsString
    Rectangle (615,500 100x20), "%.1f"", text variable: ref.parts.ron.targetOffset.arcseconds.value
    Button (615,530 100x35), "Move back to 0", input disabled if: widget.moveRelative.ronDisabled
        OnMouseClick: execute {
            ref.processes.moveRelative.request(
                units := AxesMoveUnits.DEGREES,
                azi := 0.0,
                ele := 0.0,
                rot := 0.0,
                roc := 0.0,
                ron :=  -ref.parts.ron.targetOffset.degrees.value,
                doAzi := FALSE,
                doEle := FALSE,
                doRot := FALSE,
                doRoc := FALSE,
                doRon := TRUE, preferMostTravel := widget.preferMostTravel);
        }
    Rectangle (615,480 100x40), colour toggle: widget.moveRelative.ronDisabled
    Label (555,480 60x30), "Nasmyth rotation"
    Rectangle (380,235 300x30), "Nasmyth rotation (%s)", text variable: ref.config.nasmythRotatorName
    Rectangle (380,100 305x30), "Cassegrain rotation (%s)", text variable: ref.config.cassegrainRotatorName
    Checkbox (20,60 195x30), "Prefer most travel left", variable: widget.preferMostTravel
END_VISUALIZATION

// ---- MTCS/Axes/Visu/VISU_AxesManual_Offsets_OLD.TcVIS
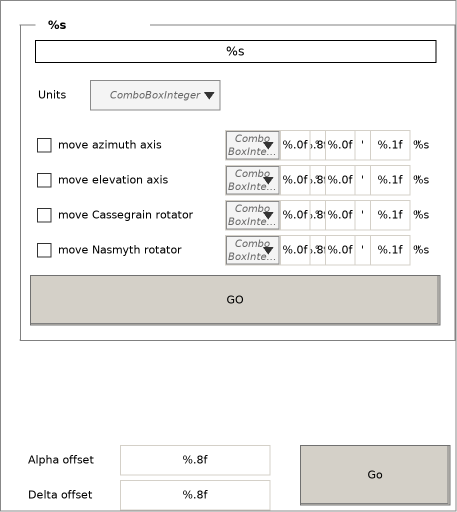
VISUALIZATION VISU_AxesManual_Offsets_OLD  // 457x512
VAR_IN_OUT
	ref : Axes;
    widget : AxesManualOffsetsWidget;
END_VAR
    Frame (15,10 440x370)
        shows VISU_AxesMultiMoveProcess(ref := ref.processes.moveRelative, widget := widget.moveRelative)
    Textfield (120,445 150x30), "%.8f", text variable: ref.processes.pointRelative.set.alpha
        OnMouseClick: write the text variable via VisuDialogs.Numpad
    Label (25,445 100x30), "Alpha offset"
    Textfield (120,480 150x30), "%.8f", text variable: ref.processes.pointRelative.set.delta
        OnMouseClick: write the text variable via VisuDialogs.Numpad
    Label (25,480 100x30), "Delta offset"
    Button (300,445 150x60), "Go", input disabled if: ref.processes.pointRelative.statuses.enabledStatus.disabled
        OnMouseClick: execute { ref.processes.pointRelative.do_request := TRUE; }
END_VISUALIZATION

// ---- MTCS/Axes/Visu/VISU_AxesRotationAxis_Processes.TcVIS
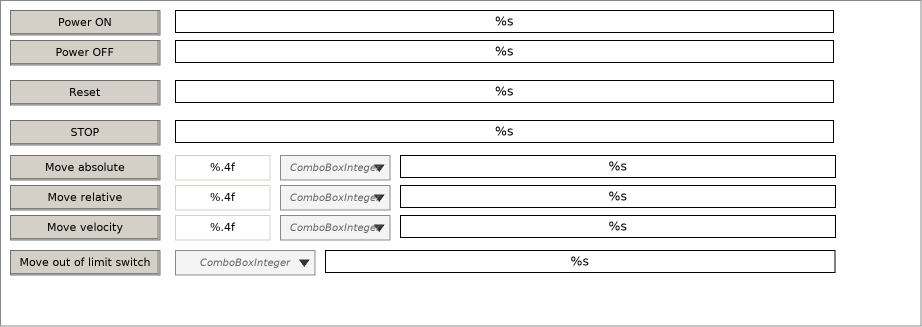
VISUALIZATION VISU_AxesRotationAxis_Processes  // 922x327
VAR_IN_OUT
	ref : AxesRotationAxis;
    ref_driveChannel : AX52XXDriveChannel;
    widget : AxesRotationAxisWidget;
END_VAR
    Frame (10,10 910x55)
        shows VISU_Axes_Commands_Power(powerOn := ref.processes.powerOn, powerOff := ref.processes.powerOff, powerOnStatus := widget.processes_powerOnStatus, powerOffStatus := widget.processes_powerOffStatus)
    Frame (10,80 910x25)
        shows VISU_Axes_Commands_Reset(reset := ref.processes.reset, resetStatus := widget.processes_resetStatus)
    Frame (10,120 910x205)
        shows VISU_Axes_Commands_Movement(stop := ref.processes.stop, moveOutOfLimitSwitch := ref.processes.moveOutOfLimitSwitch, moveAbsolute := ref.processes.moveAbsolute, moveRelative := ref.processes.moveRelative, moveVelocity := ref.processes.moveVelocity, stopStatus := widget.processes_stopStatus, moveOutOfLimitSwitchStatus := widget.processes_moveOutOfLimitSwitchStatus, moveAbsoluteStatus := widget.processes_moveAbsoluteStatus, moveRelativeStatus := widget.processes_moveRelativeStatus, moveVelocityStatus := widget.processes_moveVelocityStatus)
END_VISUALIZATION

// ---- MTCS/Axes/Visu/VISU_AxesRotationAxis_Overview.TcVIS
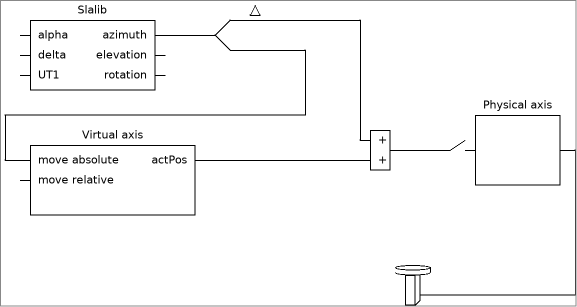
VISUALIZATION VISU_AxesRotationAxis_Overview  // 577x307
VAR_IN_OUT
	ref : AxesRotationAxis;
    widget : AxesRotationAxisWidget;
END_VAR
    Rectangle (405,275 10x30)
    Rectangle (30,20 125x70)
    Line (20,35) (30,35)
    Label (35,25 50x20), "alpha"
    Line (20,55) (30,55)
    Label (35,45 50x20), "delta"
    Line (20,75) (30,75)
    Label (35,65 50x20), "UT1"
    Polyline (255,5) (250,15) (260,15) (255,5)
    Label (30,0 125x20), "Slalib"
    Label (95,25 55x20), "azimuth"
    Label (90,45 60x20), "elevation"
    Label (100,65 50x20), "rotation"
    Line (155,55) (165,55)
    Line (155,75) (165,75)
    Rectangle (30,145 165x70)
    Label (35,150 95x20), "move absolute"
    Line (20,180) (30,180)
    Label (35,170 85x20), "move relative"
    Label (30,125 165x20), "Virtual axis"
    Label (135,150 55x20), "actPos"
    Polyline (155,35) (215,35) (230,50)
    Polyline (230,50) (305,50) (305,115) (5,115) (5,160) (30,160)
    Polyline (215,35) (230,20) (360,20) (360,140) (370,140)
    Polyline (195,160) (370,160)
    Rectangle (370,130 20x40)
    Label (375,130 15x20), "+"
    Label (375,150 15x20), "+"
    Line (390,150) (450,150)
    Line (450,150) (465,140)
    Line (465,150) (475,150)
    Rectangle (475,115 85x70)
    Label (475,95 85x20), "Physical axis"
    Polyline (560,150) (575,150) (575,295) (420,295)
    Polyline (415,305) (420,300) (420,275)
    Ellipse (395,270 35x5)
    Rectangle (395,270 35x2)
    Ellipse (395,265 35x5)
    Line (430,267) (430,272)
END_VISUALIZATION

// ---- MTCS/Axes/Visu/VISU_AxesElevationAxis_Processes.TcVIS
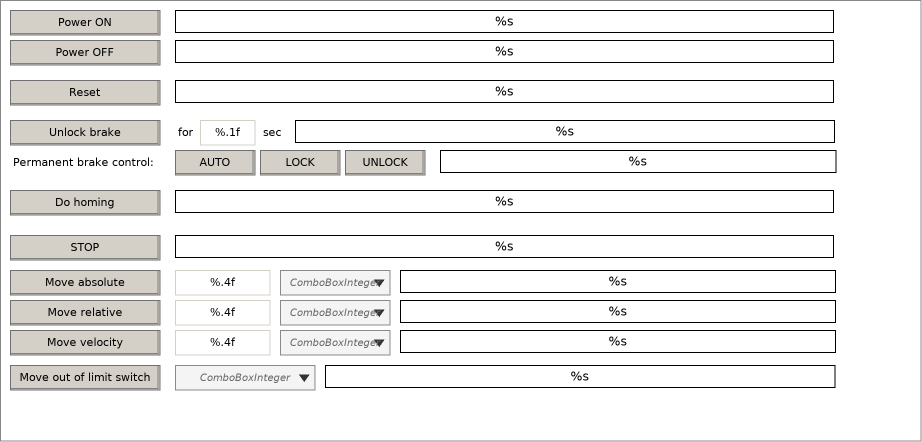
VISUALIZATION VISU_AxesElevationAxis_Processes  // 922x442
VAR_IN_OUT
	ref : AxesElevationAxis;
    ref_driveChannel : AX52XXDriveChannel;
    widget : AxesElevationAxisWidget;
END_VAR
    Frame (10,10 910x55)
        shows VISU_Axes_Commands_Power(powerOn := ref.processes.powerOn, powerOff := ref.processes.powerOff, powerOnStatus := widget.processes_powerOnStatus, powerOffStatus := widget.processes_powerOffStatus)
    Frame (10,80 910x25)
        shows VISU_Axes_Commands_Reset(reset := ref.processes.reset, resetStatus := widget.processes_resetStatus)
    Frame (10,120 910x55)
        shows VISU_Axes_Commands_Brake(unlockBrake := ref.processes.unlockBrake, setBrake := ref_driveChannel.processes.setBrake, unlockBrakeStatus := widget.processes_unlockBrakeStatus, setBrakeStatus := widget.driveChannel.processes_setBrakeStatus)
    Frame (10,190 910x35)
        shows VISU_Axes_Commands_DoHoming(doHoming := ref.processes.doHoming, doHomingStatus := widget.processes_doHomingStatus)
    Frame (10,235 910x205)
        shows VISU_Axes_Commands_Movement(stop := ref.processes.stop, moveOutOfLimitSwitch := ref.processes.moveOutOfLimitSwitch, moveAbsolute := ref.processes.moveAbsolute, moveRelative := ref.processes.moveRelative, moveVelocity := ref.processes.moveVelocity, stopStatus := widget.processes_stopStatus, moveOutOfLimitSwitchStatus := widget.processes_moveOutOfLimitSwitchStatus, moveAbsoluteStatus := widget.processes_moveAbsoluteStatus, moveRelativeStatus := widget.processes_moveRelativeStatus, moveVelocityStatus := widget.processes_moveVelocityStatus)
END_VISUALIZATION

// ---- MTCS/Axes/Visu/VISU_AxesManual_MoveVelocity.TcVIS
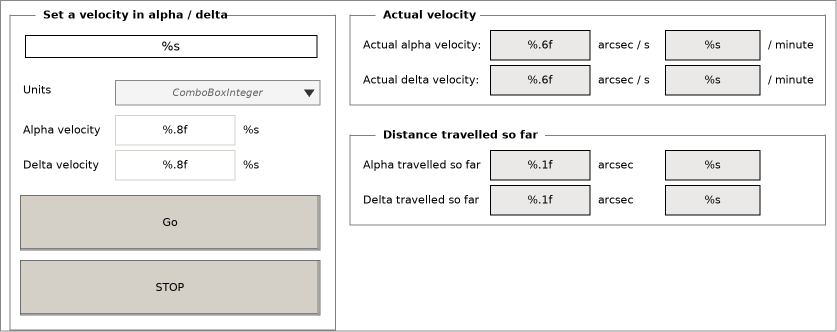
VISUALIZATION VISU_AxesManual_MoveVelocity  // 837x332
VAR_IN_OUT
	ref : Axes;
    widget : AxesManualMoveVelocityWidget;
END_VAR
    Polyline (225,15) (335,15) (335,330) (10,330) (10,15) (35,15)
    Polyline (480,15) (825,15) (825,105) (350,105) (350,15) (375,15)
    Label (380,5 100x20), "Actual velocity"
    Label (380,125 155x20), "Distance travelled so far"
    Polyline (545,135) (825,135) (825,225) (350,225) (350,135) (375,135)
    Textfield (115,115 120x30), "%.8f", text variable: widget.field_alphaVelocity
        OnMouseClick: write the text variable via VisuDialogs.Numpad
    Label (20,115 95x30), "Alpha velocity"
    Textfield (115,150 120x30), "%.8f", text variable: widget.field_deltaVelocity
        OnMouseClick: write the text variable via VisuDialogs.Numpad
    Label (20,150 95x30), "Delta velocity"
    Button (20,195 300x55), "Go", input disabled if: ref.processes.setAlphaDeltaVelocity.statuses.enabledStatus.disabled
        OnMouseClick: execute { widget.do_start := TRUE; }
    ComboBoxInteger (115,80 205x25), variable: widget.field_units, text list: 'AxesMoveVelocityUnitsTextList'
    Frame (25,35 295x25)
        shows VISU_StatusWidget(widget := widget.setAlphaDeltaVelocityStatus)
    Label (20,75 95x30), "Units"
    Rectangle (240,115 80x30), "%s", text variable: widget.label_units
    Label (360,30 145x30), "Actual alpha velocity:"
    Label (360,65 145x30), "Actual delta velocity:"
    Rectangle (490,30 100x30), "%.6f", text variable: ref.target.alphaVelocity.arcsecondsPerSecond.value
    Rectangle (490,65 100x30), "%.6f", text variable: ref.target.deltaVelocity.arcsecondsPerSecond.value
    Label (595,30 65x30), "arcsec / s"
    Rectangle (665,30 95x30), "%s", text variable: widget.alphaPerMinute.hmsString
    Rectangle (665,65 95x30), "%s", text variable: widget.deltaPerMinute.dmsString
    Label (765,30 70x30), "/ minute"
    Label (360,185 145x30), "Delta travelled so far"
    Label (360,150 145x30), "Alpha travelled so far"
    Rectangle (490,150 100x30), "%.1f", text variable: ref.target.alphaTravelled.arcseconds.value
    Rectangle (490,185 100x30), "%.1f", text variable: ref.target.deltaTravelled.arcseconds.value
    Label (595,150 75x30), "arcsec"
    Label (595,65 65x30), "arcsec / s"
    Label (765,65 70x30), "/ minute"
    Label (595,185 75x30), "arcsec"
    Rectangle (665,185 95x30), "%s", text variable: widget.deltaTravelledSoFar.dmsString
    Rectangle (665,150 95x30), "%s", text variable: widget.alphaTravelledSoFar.hmsString
    Button (20,260 300x55), "STOP", input disabled if: ref.processes.setAlphaDeltaVelocity.statuses.enabledStatus.disabled
        OnMouseClick: execute { widget.do_stop := TRUE; }
    Rectangle (240,150 80x30), "%s", text variable: widget.label_units
    Label (40,5 180x20), "Set a velocity in alpha / delta"
END_VISUALIZATION

// ---- MTCS/Axes/Visu/VISU_AxesManual_Offsets_AziEleRot.TcVIS
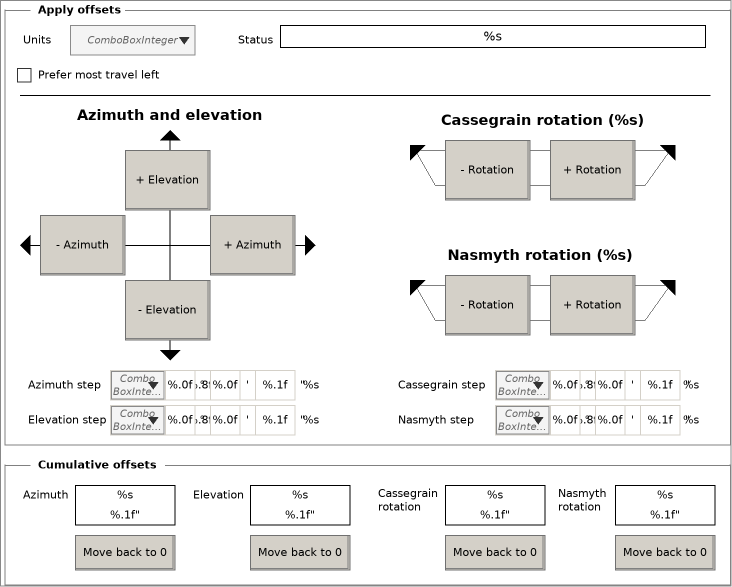
VISUALIZATION VISU_AxesManual_Offsets_AziEleRot  // 732x587
VAR_IN_OUT
	ref : Axes;
    widget : AxesManualOffsetsWidget;
END_VAR
    Polyline (125,10) (730,10) (730,445) (5,445) (5,10) (30,10)
    Polygon (670,150) (645,185) (435,185) (415,150)
    Line (170,355) (170,135)
    Line (25,245) (315,245)
    ComboBoxInteger (70,25 125x30), variable: widget.moveRelative.units, text list: 'AxesMoveProcessUnitsTextList'
    Rectangle (300,370 35x30), "%s", text variable: widget.moveRelative.unitsText, invisible if: widget.moveRelative.units = AxesMoveProcessWidgetUnits.DEGMINSEC
    Textfield (110,370 180x30), "%.8f", text variable: widget.moveRelative.field_azi_decimal, invisible if: widget.moveRelative.units = AxesMoveProcessWidgetUnits.DEGMINSEC, input disabled if: widget.moveRelative.aziDisabled
        OnMouseClick: write the text variable via VisuDialogs.Numpad
    Textfield (165,370 30x30), "%.0f", text variable: widget.moveRelative.field_azi_d, invisible if: widget.moveRelative.units <> AxesMoveProcessWidgetUnits.DEGMINSEC, input disabled if: widget.moveRelative.aziDisabled
        OnMouseClick: write the text variable via VisuDialogs.Numpad
    ComboBoxInteger (111,371 53x28), variable: widget.moveRelative.field_azi_sign, invisible if: widget.moveRelative.units <> AxesMoveProcessWidgetUnits.DEGMINSEC, input disabled if: widget.moveRelative.aziDisabled, text list: 'AxesDialogSignTextList'
    Textfield (210,370 30x30), "%.0f", text variable: widget.moveRelative.field_azi_m, invisible if: widget.moveRelative.units <> AxesMoveProcessWidgetUnits.DEGMINSEC, input disabled if: widget.moveRelative.aziDisabled
        OnMouseClick: write the text variable via VisuDialogs.Numpad
    Textfield (255,370 40x30), "%.1f", text variable: widget.moveRelative.field_azi_s, invisible if: widget.moveRelative.units <> AxesMoveProcessWidgetUnits.DEGMINSEC, input disabled if: widget.moveRelative.aziDisabled
        OnMouseClick: write the text variable via VisuDialogs.Numpad
    Label (195,370 15x30), "°", invisible if: widget.moveRelative.units <> AxesMoveProcessWidgetUnits.DEGMINSEC
    Label (240,370 15x30), "'", invisible if: widget.moveRelative.units <> AxesMoveProcessWidgetUnits.DEGMINSEC
    Label (295,370 15x30), """, invisible if: widget.moveRelative.units <> AxesMoveProcessWidgetUnits.DEGMINSEC
    Rectangle (300,405 35x30), "%s", text variable: widget.moveRelative.unitsText, invisible if: widget.moveRelative.units = AxesMoveProcessWidgetUnits.DEGMINSEC
    Textfield (110,405 180x30), "%.8f", text variable: widget.moveRelative.field_ele_decimal, invisible if: widget.moveRelative.units = AxesMoveProcessWidgetUnits.DEGMINSEC, input disabled if: widget.moveRelative.eleDisabled
        OnMouseClick: write the text variable via VisuDialogs.Numpad
    Textfield (165,405 30x30), "%.0f", text variable: widget.moveRelative.field_ele_d, invisible if: widget.moveRelative.units <> AxesMoveProcessWidgetUnits.DEGMINSEC, input disabled if: widget.moveRelative.eleDisabled
        OnMouseClick: write the text variable via VisuDialogs.Numpad
    ComboBoxInteger (111,406 53x28), variable: widget.moveRelative.field_ele_sign, invisible if: widget.moveRelative.units <> AxesMoveProcessWidgetUnits.DEGMINSEC, input disabled if: widget.moveRelative.eleDisabled, text list: 'AxesDialogSignTextList'
    Textfield (210,405 30x30), "%.0f", text variable: widget.moveRelative.field_ele_m, invisible if: widget.moveRelative.units <> AxesMoveProcessWidgetUnits.DEGMINSEC, input disabled if: widget.moveRelative.eleDisabled
        OnMouseClick: write the text variable via VisuDialogs.Numpad
    Textfield (255,405 40x30), "%.1f", text variable: widget.moveRelative.field_ele_s, invisible if: widget.moveRelative.units <> AxesMoveProcessWidgetUnits.DEGMINSEC, input disabled if: widget.moveRelative.eleDisabled
        OnMouseClick: write the text variable via VisuDialogs.Numpad
    Label (195,405 15x30), "°", invisible if: widget.moveRelative.units <> AxesMoveProcessWidgetUnits.DEGMINSEC
    Label (240,405 15x30), "'", invisible if: widget.moveRelative.units <> AxesMoveProcessWidgetUnits.DEGMINSEC
    Label (295,405 15x30), """, invisible if: widget.moveRelative.units <> AxesMoveProcessWidgetUnits.DEGMINSEC
    Rectangle (680,370 35x30), "%s", text variable: widget.moveRelative.unitsText, invisible if: widget.moveRelative.units = AxesMoveProcessWidgetUnits.DEGMINSEC
    Textfield (495,370 180x30), "%.8f", text variable: widget.moveRelative.field_roc_decimal, invisible if: widget.moveRelative.units = AxesMoveProcessWidgetUnits.DEGMINSEC, input disabled if: widget.moveRelative.rocDisabled
        OnMouseClick: write the text variable via VisuDialogs.Numpad
    Textfield (550,370 30x30), "%.0f", text variable: widget.moveRelative.field_roc_d, invisible if: widget.moveRelative.units <> AxesMoveProcessWidgetUnits.DEGMINSEC, input disabled if: widget.moveRelative.rocDisabled
        OnMouseClick: write the text variable via VisuDialogs.Numpad
    ComboBoxInteger (496,371 53x28), variable: widget.moveRelative.field_roc_sign, invisible if: widget.moveRelative.units <> AxesMoveProcessWidgetUnits.DEGMINSEC, input disabled if: widget.moveRelative.rocDisabled, text list: 'AxesDialogSignTextList'
    Textfield (595,370 30x30), "%.0f", text variable: widget.moveRelative.field_roc_m, invisible if: widget.moveRelative.units <> AxesMoveProcessWidgetUnits.DEGMINSEC, input disabled if: widget.moveRelative.rocDisabled
        OnMouseClick: write the text variable via VisuDialogs.Numpad
    Textfield (640,370 40x30), "%.1f", text variable: widget.moveRelative.field_roc_s, invisible if: widget.moveRelative.units <> AxesMoveProcessWidgetUnits.DEGMINSEC, input disabled if: widget.moveRelative.rocDisabled
        OnMouseClick: write the text variable via VisuDialogs.Numpad
    Label (580,370 15x30), "°", invisible if: widget.moveRelative.units <> AxesMoveProcessWidgetUnits.DEGMINSEC
    Label (625,370 15x30), "'", invisible if: widget.moveRelative.units <> AxesMoveProcessWidgetUnits.DEGMINSEC
    Label (680,370 15x30), """, invisible if: widget.moveRelative.units <> AxesMoveProcessWidgetUnits.DEGMINSEC
    Rectangle (680,405 35x30), "%s", text variable: widget.moveRelative.unitsText, invisible if: widget.moveRelative.units = AxesMoveProcessWidgetUnits.DEGMINSEC
    Textfield (495,405 180x30), "%.8f", text variable: widget.moveRelative.field_ron_decimal, invisible if: widget.moveRelative.units = AxesMoveProcessWidgetUnits.DEGMINSEC, input disabled if: widget.moveRelative.ronDisabled
        OnMouseClick: write the text variable via VisuDialogs.Numpad
    Textfield (550,405 30x30), "%.0f", text variable: widget.moveRelative.field_ron_d, invisible if: widget.moveRelative.units <> AxesMoveProcessWidgetUnits.DEGMINSEC, input disabled if: widget.moveRelative.ronDisabled
        OnMouseClick: write the text variable via VisuDialogs.Numpad
    ComboBoxInteger (496,406 53x28), variable: widget.moveRelative.field_ron_sign, invisible if: widget.moveRelative.units <> AxesMoveProcessWidgetUnits.DEGMINSEC, input disabled if: widget.moveRelative.ronDisabled, text list: 'AxesDialogSignTextList'
    Textfield (595,405 30x30), "%.0f", text variable: widget.moveRelative.field_ron_m, invisible if: widget.moveRelative.units <> AxesMoveProcessWidgetUnits.DEGMINSEC, input disabled if: widget.moveRelative.ronDisabled
        OnMouseClick: write the text variable via VisuDialogs.Numpad
    Textfield (640,405 40x30), "%.1f", text variable: widget.moveRelative.field_ron_s, invisible if: widget.moveRelative.units <> AxesMoveProcessWidgetUnits.DEGMINSEC, input disabled if: widget.moveRelative.ronDisabled
        OnMouseClick: write the text variable via VisuDialogs.Numpad
    Label (580,405 15x30), "°", invisible if: widget.moveRelative.units <> AxesMoveProcessWidgetUnits.DEGMINSEC
    Label (625,405 15x30), "'", invisible if: widget.moveRelative.units <> AxesMoveProcessWidgetUnits.DEGMINSEC
    Label (680,405 15x30), """, invisible if: widget.moveRelative.units <> AxesMoveProcessWidgetUnits.DEGMINSEC
    Frame (280,25 430x25)
        shows VISU_StatusWidget(widget := widget.moveRelative.actualStatus)
    Label (35,0 100x20), "Apply offsets"
    Button (125,150 85x60), "+ Elevation", input disabled if: widget.moveRelative.eleDisabled
        OnMouseClick: execute {
            ref.processes.moveRelative.request(
                units := AxesMoveUnits.DEGREES,
                azi := 0.0,
                ele := widget.moveRelative.eleDeg,
                rot := 0.0,
                roc := 0.0,
                ron := 0.0,
                doAzi := FALSE,
                doEle := TRUE,
                doRot := FALSE,
                doRoc := FALSE,
                doRon := FALSE,
                preferMostTravel := widget.preferMostTravel);
        }
    Button (125,280 85x60), "- Elevation", input disabled if: widget.moveRelative.eleDisabled
        OnMouseClick: execute {
            ref.processes.moveRelative.request(
                units := AxesMoveUnits.DEGREES,
                azi := 0.0,
                ele := -widget.moveRelative.eleDeg,
                rot := 0.0,
                roc := 0.0,
                ron := 0.0,
                doAzi := FALSE,
                doEle := TRUE,
                doRot := FALSE,
                doRoc := FALSE,
                doRon := FALSE,
                preferMostTravel := widget.preferMostTravel);
        }
    Button (210,215 85x60), "+ Azimuth", input disabled if: widget.moveRelative.aziDisabled
        OnMouseClick: execute {
            ref.processes.moveRelative.request(
                units := AxesMoveUnits.DEGREES,
                azi := widget.moveRelative.aziDeg,
                ele := 0.0,
                rot := 0.0,
                roc := 0.0,
                ron := 0.0,
                doAzi := TRUE,
                doEle := FALSE,
                doRot := FALSE,
                doRoc := FALSE,
                doRon := FALSE,
                preferMostTravel := widget.preferMostTravel);
        }
    Button (40,215 85x60), "- Azimuth", input disabled if: widget.moveRelative.aziDisabled
        OnMouseClick: execute {
            ref.processes.moveRelative.request(
                units := AxesMoveUnits.DEGREES,
                azi := -widget.moveRelative.aziDeg,
                ele := 0.0,
                rot := 0.0,
                roc := 0.0,
                ron := 0.0,
                doAzi := TRUE,
                doEle := FALSE,
                doRot := FALSE,
                doRoc := FALSE,
                doRon := FALSE,
                preferMostTravel := widget.preferMostTravel);
        }
    Label (25,370 80x30), "Azimuth step"
    Label (25,405 85x30), "Elevation step"
    Button (550,140 85x60), "+ Rotation", input disabled if: widget.moveRelative.rocDisabled
        OnMouseClick: execute {
            ref.processes.moveRelative.request(
                units := AxesMoveUnits.DEGREES,
                azi := 0.0,
                ele := 0.0,
                rot := 0.0,
                roc := widget.moveRelative.rocDeg,
                ron := 0.0,
                doAzi := FALSE,
                doEle := FALSE,
                doRot := FALSE,
                doRoc := TRUE,
                doRon := FALSE,
                preferMostTravel := widget.preferMostTravel);
        }
    Button (445,140 85x60), "- Rotation", input disabled if: widget.moveRelative.rocDisabled
        OnMouseClick: execute {
            ref.processes.moveRelative.request(
                units := AxesMoveUnits.DEGREES,
                azi := 0.0,
                ele := 0.0,
                rot := 0.0,
                roc := -widget.moveRelative.rocDeg,
                ron := 0.0,
                doAzi := FALSE,
                doEle := FALSE,
                doRot := FALSE,
                doRoc := TRUE,
                doRon := FALSE,
                preferMostTravel := widget.preferMostTravel);
        }
    Polygon (160,140) (170,130) (180,140)
    Polygon (30,255) (20,245) (30,235)
    Polygon (305,255) (315,245) (305,235)
    Polygon (160,350) (170,360) (180,350)
    Polygon (675,160) (675,145) (660,145)
    Polygon (410,160) (425,145) (410,145)
    Label (395,370 130x30), "Cassegrain step"
    Label (395,405 130x30), "Nasmyth step"
    Label (20,25 55x30), "Units"
    Label (235,25 45x30), "Status"
    Line (20,95) (710,95)
    Polygon (670,285) (645,320) (435,320) (415,285)
    Button (550,275 85x60), "+ Rotation", input disabled if: widget.moveRelative.ronDisabled
        OnMouseClick: execute {
            ref.processes.moveRelative.request(
                units := AxesMoveUnits.DEGREES,
                azi := 0.0,
                ele := 0.0,
                rot := 0.0,
                roc := 0.0,
                ron := widget.moveRelative.ronDeg,
                doAzi := FALSE,
                doEle := FALSE,
                doRot := FALSE,
                doRoc := FALSE,
                doRon := TRUE,
                preferMostTravel := widget.preferMostTravel);
        }
    Button (445,275 85x60), "- Rotation", input disabled if: widget.moveRelative.ronDisabled
        OnMouseClick: execute {
            ref.processes.moveRelative.request(
                units := AxesMoveUnits.DEGREES,
                azi := 0.0,
                ele := 0.0,
                rot := 0.0,
                roc := 0.0,
                ron := -widget.moveRelative.ronDeg,
                doAzi := FALSE,
                doEle := FALSE,
                doRot := FALSE,
                doRoc := FALSE,
                doRon := TRUE,
                preferMostTravel := widget.preferMostTravel);
        }
    Polygon (675,295) (675,280) (660,280)
    Polygon (410,295) (425,280) (410,280)
    Label (35,100 270x30), "Azimuth and elevation"
    Polyline (165,465) (730,465) (730,585) (5,585) (5,465) (30,465)
    Rectangle (75,485 100x20), "%s", text variable: widget.aziTargetOffset.dmsString
    Rectangle (75,505 100x20), "%.1f"", text variable: ref.parts.azi.targetOffset.arcseconds.value
    Button (75,535 100x35), "Move back to 0", input disabled if: widget.moveRelative.aziDisabled
        OnMouseClick: execute {
            ref.processes.moveRelative.request(
                units := AxesMoveUnits.DEGREES,
                azi := -ref.parts.azi.targetOffset.degrees.value,
                ele := 0.0,
                rot := 0.0,
                roc := 0.0,
                ron := 0.0,
                doAzi := TRUE,
                doEle := FALSE,
                doRot := FALSE,
                doRoc := FALSE,
                doRon := FALSE,
                preferMostTravel := widget.preferMostTravel);
        }
    Label (35,455 120x20), "Cumulative offsets"
    Rectangle (75,485 100x40), colour toggle: widget.moveRelative.aziDisabled
    Rectangle (250,485 100x20), "%s", text variable: widget.eleTargetOffset.dmsString
    Rectangle (250,505 100x20), "%.1f"", text variable: ref.parts.ele.targetOffset.arcseconds.value
    Button (250,535 100x35), "Move back to 0", input disabled if: widget.moveRelative.eleDisabled
        OnMouseClick: execute {
            ref.processes.moveRelative.request(
                units := AxesMoveUnits.DEGREES,
                azi := 0.0,
                ele := -ref.parts.ele.targetOffset.degrees.value,
                rot := 0.0,
                roc := 0.0,
                ron := 0.0,
                doAzi := FALSE,
                doEle := TRUE,
                doRot := FALSE,
                doRoc := FALSE,
                doRon := FALSE,
                preferMostTravel := widget.preferMostTravel);
        }
    Rectangle (250,485 100x40), colour toggle: widget.moveRelative.eleDisabled
    Rectangle (445,485 100x20), "%s", text variable: widget.rocTargetOffset.dmsString
    Rectangle (445,505 100x20), "%.1f"", text variable: ref.parts.roc.targetOffset.arcseconds.value
    Button (445,535 100x35), "Move back to 0", input disabled if: widget.moveRelative.rocDisabled
        OnMouseClick: execute {
            ref.processes.moveRelative.request(
                units := AxesMoveUnits.DEGREES,
                azi := 0.0,
                ele := 0.0,
                rot := 0.0,
                roc := -ref.parts.roc.targetOffset.degrees.value,
                ron := 0.0,
                doAzi := FALSE,
                doEle := FALSE,
                doRot := FALSE,
                doRoc := TRUE,
                doRon := FALSE,
                preferMostTravel := widget.preferMostTravel);
        }
    Rectangle (445,485 100x40), colour toggle: widget.moveRelative.rocDisabled
    Label (375,485 70x30), "Cassegrain rotation"
    Rectangle (615,485 100x20), "%s", text variable: widget.ronTargetOffset.dmsString
    Rectangle (615,505 100x20), "%.1f"", text variable: ref.parts.ron.targetOffset.arcseconds.value
    Button (615,535 100x35), "Move back to 0", input disabled if: widget.moveRelative.ronDisabled
        OnMouseClick: execute {
            ref.processes.moveRelative.request(
                units := AxesMoveUnits.DEGREES,
                azi := 0.0,
                ele := 0.0,
                rot := 0.0,
                roc := 0.0,
                ron :=  -ref.parts.ron.targetOffset.degrees.value,
                doAzi := FALSE,
                doEle := FALSE,
                doRot := FALSE,
                doRoc := FALSE,
                doRon := TRUE, preferMostTravel := widget.preferMostTravel);
        }
    Rectangle (615,485 100x40), colour toggle: widget.moveRelative.ronDisabled
    Label (555,485 60x30), "Nasmyth rotation"
    Label (20,485 55x20), "Azimuth"
    Label (190,485 55x20), "Elevation"
    Rectangle (390,240 300x30), "Nasmyth rotation (%s)", text variable: ref.config.nasmythRotatorName
    Rectangle (390,105 305x30), "Cassegrain rotation (%s)", text variable: ref.config.cassegrainRotatorName
    Checkbox (15,60 195x30), "Prefer most travel left", variable: widget.preferMostTravel
END_VISUALIZATION

// ---- MTCS/Axes/Visu/VISU_AxesManual_Joystick_AziEle.TcVIS
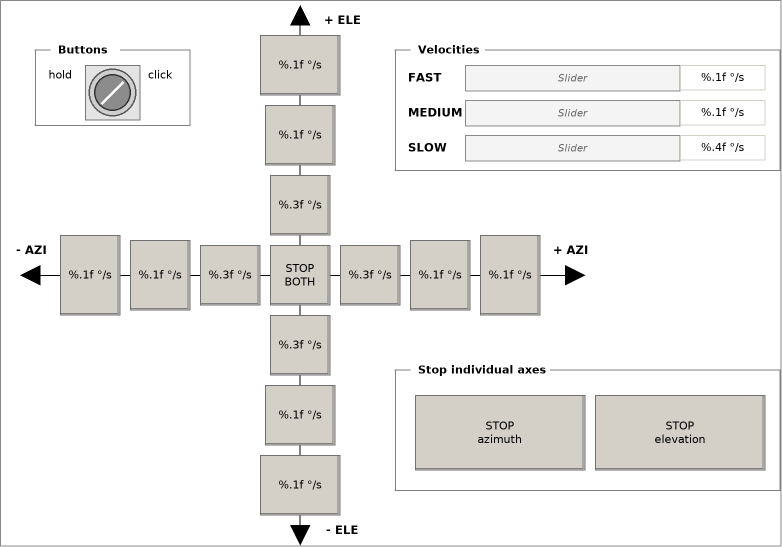
VISUALIZATION VISU_AxesManual_Joystick_AziEle  // 782x547
VAR_IN_OUT
	ref : Axes;
    widget : AxesManualJoystickAziEleWidget;
END_VAR
    Polyline (410,50) (395,50) (395,170) (780,170) (780,50) (485,50)
    Line (40,275) (575,275)
    Line (300,525) (300,25)
    Slider (465,65 215x26), variable: widget.joystick_velocity_fast, input disabled if: widget.joystick_disabled, scale 0..3
    Button (260,35 80x60), "%.1f °/s", text variable: widget.joystick_velocity_fast, input disabled if: widget.jog_ele_disabled
        tap widget.jog_ele_forward_fast
    Button (265,105 70x60), "%.1f °/s", text variable: widget.joystick_velocity_medium, input disabled if: widget.jog_ele_disabled
        tap widget.jog_ele_forward_medium
    Button (270,175 60x60), "%.3f °/s", text variable: widget.joystick_velocity_slow, input disabled if: widget.jog_ele_disabled
        tap widget.jog_ele_forward_slow
    Button (270,245 60x60), "STOP BOTH", input disabled if: ref.processes.stop.statuses.enabledStatus.disabled
        OnMouseClick: execute { ref.processes.stop.request(); }
    Button (260,455 80x60), "%.1f °/s", text variable: widget.joystick_velocity_fast, input disabled if: widget.jog_ele_disabled
        tap widget.jog_ele_backwards_fast
    Button (265,385 70x60), "%.1f °/s", text variable: widget.joystick_velocity_medium, input disabled if: widget.jog_ele_disabled
        tap widget.jog_ele_backwards_medium
    Button (270,315 60x60), "%.3f °/s", text variable: widget.joystick_velocity_slow, input disabled if: widget.jog_ele_disabled
        tap widget.jog_ele_backwards_slow
    Button (200,245 60x60), "%.3f °/s", text variable: widget.joystick_velocity_slow, input disabled if: widget.jog_azi_disabled
        tap widget.jog_azi_backwards_slow
    Button (130,240 60x70), "%.1f °/s", text variable: widget.joystick_velocity_medium, input disabled if: widget.jog_azi_disabled
        tap widget.jog_azi_backwards_medium
    Button (60,235 60x80), "%.1f °/s", text variable: widget.joystick_velocity_fast, input disabled if: widget.jog_azi_disabled
        tap widget.jog_azi_backwards_fast
    Button (480,235 60x80), "%.1f °/s", text variable: widget.joystick_velocity_fast, input disabled if: widget.jog_azi_disabled
        tap widget.jog_azi_forward_fast
    Button (410,240 60x70), "%.1f °/s", text variable: widget.joystick_velocity_medium, input disabled if: widget.jog_azi_disabled
        tap widget.jog_azi_forward_medium
    Button (340,245 60x60), "%.3f °/s", text variable: widget.joystick_velocity_slow, input disabled if: widget.jog_azi_disabled
        tap widget.jog_azi_forward_slow
    Textfield (680,65 85x25), "%.1f °/s", text variable: widget.joystick_velocity_fast, input disabled if: widget.joystick_disabled
        OnMouseClick: write the text variable via VisuDialogs.Numpad, min 0, max 3
    Polygon (290,25) (300,5) (310,25)
    Polygon (290,525) (300,545) (310,525)
    Polygon (565,285) (565,265) (585,275)
    Polygon (40,285) (40,265) (20,275)
    Label (405,65 70x25), "FAST"
    Slider (465,100 215x26), variable: widget.joystick_velocity_medium, input disabled if: widget.joystick_disabled, scale 0..3
    Label (405,100 70x25), "MEDIUM"
    Slider (465,135 215x26), variable: widget.joystick_velocity_slow, input disabled if: widget.joystick_disabled, scale 0..3
    Label (405,135 70x25), "SLOW"
    Label (415,40 70x20), "Velocities"
    Textfield (680,100 85x25), "%.1f °/s", text variable: widget.joystick_velocity_medium, input disabled if: widget.joystick_disabled
        OnMouseClick: write the text variable via VisuDialogs.Numpad, min 0, max 3
    Textfield (680,135 85x25), "%.4f °/s", text variable: widget.joystick_velocity_slow, input disabled if: widget.joystick_disabled
        OnMouseClick: write the text variable via VisuDialogs.Numpad, min 0, max 3
    Label (315,5 55x30), "+ ELE"
    Label (315,515 55x30), "- ELE"
    Label (550,235 45x30), "+ AZI"
    Label (10,235 40x30), "- AZI"
    Label (415,360 135x20), "Stop individual axes"
    Polyline (410,370) (395,370) (395,490) (780,490) (780,370) (550,370)
    Button (415,395 170x75), "STOP azimuth", input disabled if: ref.parts.azi.processes.stop.statuses.enabledStatus.disabled
        OnMouseClick: execute { ref.parts.azi.processes.stop.request(); }
    Button (595,395 170x75), "STOP elevation", input disabled if: ref.parts.ele.processes.stop.statuses.enabledStatus.disabled
        OnMouseClick: execute { ref.parts.ele.processes.stop.request(); }
    Polyline (50,50) (35,50) (35,125) (190,125) (190,50) (120,50)
    RotarySwitch (85,65 55x55), variable: widget.joystick_hold, input disabled if: widget.joystick_disabled, behaviour: TOGGLE, style: Switch-RotarySwitch-Gray
    Label (145,65 50x20), "click"
    Label (35,65 40x20), "hold"
    Label (55,40 65x20), "Buttons"
END_VISUALIZATION

// ---- MTCS/Axes/Visu/VISU_AxesManual_Joystick_Rot.TcVIS
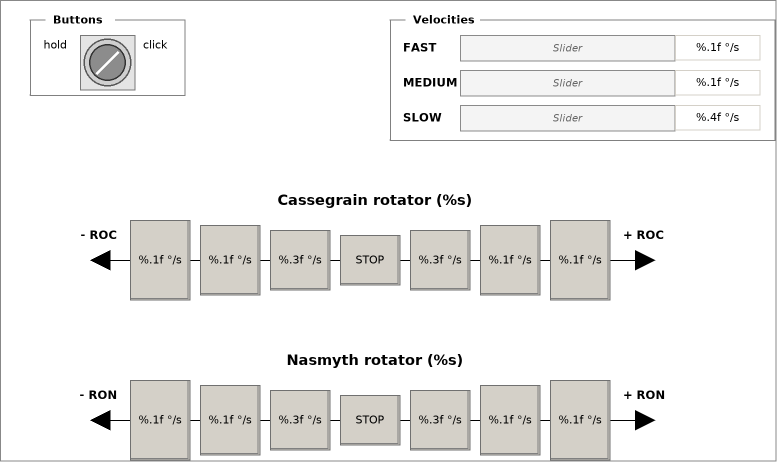
VISUALIZATION VISU_AxesManual_Joystick_Rot  // 777x462
VAR_IN_OUT
	ref : Axes;
    widget : AxesManualJoystickRotWidget;
END_VAR
    Polyline (405,20) (390,20) (390,140) (775,140) (775,20) (480,20)
    Line (110,260) (645,260)
    Slider (460,35 215x26), variable: widget.joystick_velocity_fast, input disabled if: widget.joystick_disabled, scale 0..3
    Button (270,230 60x60), "%.3f °/s", text variable: widget.joystick_velocity_slow, input disabled if: widget.jog_roc_disabled
        tap widget.jog_roc_backwards_slow
    Button (200,225 60x70), "%.1f °/s", text variable: widget.joystick_velocity_medium, input disabled if: widget.jog_roc_disabled
        tap widget.jog_roc_backwards_medium
    Button (130,220 60x80), "%.1f °/s", text variable: widget.joystick_velocity_fast, input disabled if: widget.jog_roc_disabled
        tap widget.jog_roc_backwards_fast
    Button (550,220 60x80), "%.1f °/s", text variable: widget.joystick_velocity_fast, input disabled if: widget.jog_roc_disabled
        tap widget.jog_roc_forward_fast
    Button (480,225 60x70), "%.1f °/s", text variable: widget.joystick_velocity_medium, input disabled if: widget.jog_roc_disabled
        tap widget.jog_roc_forward_medium
    Button (410,230 60x60), "%.3f °/s", text variable: widget.joystick_velocity_slow, input disabled if: widget.jog_roc_disabled
        tap widget.jog_roc_forward_slow
    Textfield (675,35 85x25), "%.1f °/s", text variable: widget.joystick_velocity_fast, input disabled if: widget.joystick_disabled
        OnMouseClick: write the text variable via VisuDialogs.Numpad, min 0, max 6
    Polygon (635,270) (635,250) (655,260)
    Polygon (110,270) (110,250) (90,260)
    Label (400,35 70x25), "FAST"
    Slider (460,70 215x26), variable: widget.joystick_velocity_medium, input disabled if: widget.joystick_disabled, scale 0..3
    Label (400,70 70x25), "MEDIUM"
    Slider (460,105 215x26), variable: widget.joystick_velocity_slow, input disabled if: widget.joystick_disabled, scale 0..3
    Label (400,105 70x25), "SLOW"
    Label (410,10 70x20), "Velocities"
    Textfield (675,70 85x25), "%.1f °/s", text variable: widget.joystick_velocity_medium, input disabled if: widget.joystick_disabled
        OnMouseClick: write the text variable via VisuDialogs.Numpad, min 0, max 3
    Textfield (675,105 85x25), "%.4f °/s", text variable: widget.joystick_velocity_slow, input disabled if: widget.joystick_disabled
        OnMouseClick: write the text variable via VisuDialogs.Numpad, min 0, max 3
    Label (620,220 45x30), "+ ROC"
    Label (80,220 40x30), "- ROC"
    Button (340,235 60x50), "STOP", input disabled if: widget.jog_roc_disabled
        OnMouseClick: execute { ref.parts.roc.processes.stop.request(); }
    Polyline (45,20) (30,20) (30,95) (185,95) (185,20) (115,20)
    RotarySwitch (80,35 55x55), variable: widget.joystick_hold, input disabled if: widget.joystick_disabled, behaviour: TOGGLE, style: Switch-RotarySwitch-Gray
    Label (140,35 50x20), "click"
    Label (30,35 40x20), "hold"
    Label (50,10 65x20), "Buttons"
    Line (110,420) (645,420)
    Button (270,390 60x60), "%.3f °/s", text variable: widget.joystick_velocity_slow, input disabled if: widget.jog_ron_disabled
        tap widget.jog_ron_backwards_slow
    Button (200,385 60x70), "%.1f °/s", text variable: widget.joystick_velocity_medium, input disabled if: widget.jog_ron_disabled
        tap widget.jog_ron_backwards_medium
    Button (130,380 60x80), "%.1f °/s", text variable: widget.joystick_velocity_fast, input disabled if: widget.jog_ron_disabled
        tap widget.jog_ron_backwards_fast
    Button (550,380 60x80), "%.1f °/s", text variable: widget.joystick_velocity_fast, input disabled if: widget.jog_ron_disabled
        tap widget.jog_ron_forward_fast
    Button (480,385 60x70), "%.1f °/s", text variable: widget.joystick_velocity_medium, input disabled if: widget.jog_ron_disabled
        tap widget.jog_ron_forward_medium
    Button (410,390 60x60), "%.3f °/s", text variable: widget.joystick_velocity_slow, input disabled if: widget.jog_ron_disabled
        tap widget.jog_ron_forward_slow
    Polygon (635,430) (635,410) (655,420)
    Polygon (110,430) (110,410) (90,420)
    Label (620,380 45x30), "+ RON"
    Label (80,380 40x30), "- RON"
    Button (340,395 60x50), "STOP", input disabled if: widget.jog_ron_disabled
        OnMouseClick: execute { ref.parts.ron.processes.stop.request(); }
    Rectangle (95,185 560x30), "Cassegrain rotator (%s)", text variable: ref.config.cassegrainRotatorName
    Rectangle (95,345 560x30), "Nasmyth rotator (%s)", text variable: ref.config.nasmythRotatorName
END_VISUALIZATION

// ---- MTCS/Axes/Visu/VISU_AxesManual_Positions.TcVIS
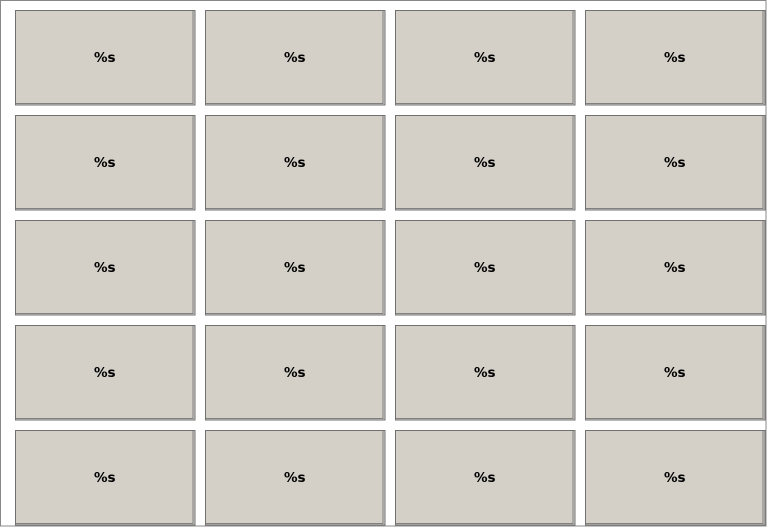
VISUALIZATION VISU_AxesManual_Positions  // 767x527
VAR_IN_OUT
	ref : Axes;
    widget : AxesManualPositionsWidget;
END_VAR
    Button (15,10 180x95), "%s", text variable: ref.config.knownPositions.position0.name, invisible if: widget.invisiblePosition0, input disabled if: ref.processes.moveKnownPosition.statuses.enabledStatus.disabled
        OnMouseClick: execute { ref.processes.moveKnownPosition.request(ref.config.knownPositions.position0.name); }
    Button (15,115 180x95), "%s", text variable: ref.config.knownPositions.position1.name, invisible if: widget.invisiblePosition1, input disabled if: ref.processes.moveKnownPosition.statuses.enabledStatus.disabled
        OnMouseClick: execute { ref.processes.moveKnownPosition.request(ref.config.knownPositions.position1.name); }
    Button (15,220 180x95), "%s", text variable: ref.config.knownPositions.position2.name, invisible if: widget.invisiblePosition2, input disabled if: ref.processes.moveKnownPosition.statuses.enabledStatus.disabled
        OnMouseClick: execute { ref.processes.moveKnownPosition.request(ref.config.knownPositions.position2.name); }
    Button (15,325 180x95), "%s", text variable: ref.config.knownPositions.position3.name, invisible if: widget.invisiblePosition3, input disabled if: ref.processes.moveKnownPosition.statuses.enabledStatus.disabled
        OnMouseClick: execute { ref.processes.moveKnownPosition.request(ref.config.knownPositions.position3.name); }
    Button (15,430 180x95), "%s", text variable: ref.config.knownPositions.position4.name, invisible if: widget.invisiblePosition4, input disabled if: ref.processes.moveKnownPosition.statuses.enabledStatus.disabled
        OnMouseClick: execute { ref.processes.moveKnownPosition.request(ref.config.knownPositions.position4.name); }
    Button (205,10 180x95), "%s", text variable: ref.config.knownPositions.position5.name, invisible if: widget.invisiblePosition5, input disabled if: ref.processes.moveKnownPosition.statuses.enabledStatus.disabled
        OnMouseClick: execute { ref.processes.moveKnownPosition.request(ref.config.knownPositions.position5.name); }
    Button (205,115 180x95), "%s", text variable: ref.config.knownPositions.position6.name, invisible if: widget.invisiblePosition6, input disabled if: ref.processes.moveKnownPosition.statuses.enabledStatus.disabled
        OnMouseClick: execute { ref.processes.moveKnownPosition.request(ref.config.knownPositions.position6.name); }
    Button (205,220 180x95), "%s", text variable: ref.config.knownPositions.position7.name, invisible if: widget.invisiblePosition7, input disabled if: ref.processes.moveKnownPosition.statuses.enabledStatus.disabled
        OnMouseClick: execute { ref.processes.moveKnownPosition.request(ref.config.knownPositions.position7.name); }
    Button (205,325 180x95), "%s", text variable: ref.config.knownPositions.position8.name, invisible if: widget.invisiblePosition8, input disabled if: ref.processes.moveKnownPosition.statuses.enabledStatus.disabled
        OnMouseClick: execute { ref.processes.moveKnownPosition.request(ref.config.knownPositions.position8.name); }
    Button (205,430 180x95), "%s", text variable: ref.config.knownPositions.position9.name, invisible if: widget.invisiblePosition9, input disabled if: ref.processes.moveKnownPosition.statuses.enabledStatus.disabled
        OnMouseClick: execute { ref.processes.moveKnownPosition.request(ref.config.knownPositions.position9.name); }
    Button (395,10 180x95), "%s", text variable: ref.config.knownPositions.position10.name, invisible if: widget.invisiblePosition10, input disabled if: ref.processes.moveKnownPosition.statuses.enabledStatus.disabled
        OnMouseClick: execute { ref.processes.moveKnownPosition.request(ref.config.knownPositions.position10.name); }
    Button (395,115 180x95), "%s", text variable: ref.config.knownPositions.position11.name, invisible if: widget.invisiblePosition11, input disabled if: ref.processes.moveKnownPosition.statuses.enabledStatus.disabled
        OnMouseClick: execute { ref.processes.moveKnownPosition.request(ref.config.knownPositions.position11.name); }
    Button (395,220 180x95), "%s", text variable: ref.config.knownPositions.position12.name, invisible if: widget.invisiblePosition12, input disabled if: ref.processes.moveKnownPosition.statuses.enabledStatus.disabled
        OnMouseClick: execute { ref.processes.moveKnownPosition.request(ref.config.knownPositions.position12.name); }
    Button (395,325 180x95), "%s", text variable: ref.config.knownPositions.position13.name, invisible if: widget.invisiblePosition13, input disabled if: ref.processes.moveKnownPosition.statuses.enabledStatus.disabled
        OnMouseClick: execute { ref.processes.moveKnownPosition.request(ref.config.knownPositions.position13.name); }
    Button (395,430 180x95), "%s", text variable: ref.config.knownPositions.position14.name, invisible if: widget.invisiblePosition14, input disabled if: ref.processes.moveKnownPosition.statuses.enabledStatus.disabled
        OnMouseClick: execute { ref.processes.moveKnownPosition.request(ref.config.knownPositions.position14.name); }
    Button (585,10 180x95), "%s", text variable: ref.config.knownPositions.position15.name, invisible if: widget.invisiblePosition15, input disabled if: ref.processes.moveKnownPosition.statuses.enabledStatus.disabled
        OnMouseClick: execute { ref.processes.moveKnownPosition.request(ref.config.knownPositions.position15.name); }
    Button (585,115 180x95), "%s", text variable: ref.config.knownPositions.position16.name, invisible if: widget.invisiblePosition16, input disabled if: ref.processes.moveKnownPosition.statuses.enabledStatus.disabled
        OnMouseClick: execute { ref.processes.moveKnownPosition.request(ref.config.knownPositions.position16.name); }
    Button (585,220 180x95), "%s", text variable: ref.config.knownPositions.position17.name, invisible if: widget.invisiblePosition17, input disabled if: ref.processes.moveKnownPosition.statuses.enabledStatus.disabled
        OnMouseClick: execute { ref.processes.moveKnownPosition.request(ref.config.knownPositions.position17.name); }
    Button (585,325 180x95), "%s", text variable: ref.config.knownPositions.position18.name, invisible if: widget.invisiblePosition18, input disabled if: ref.processes.moveKnownPosition.statuses.enabledStatus.disabled
        OnMouseClick: execute { ref.processes.moveKnownPosition.request(ref.config.knownPositions.position18.name); }
    Button (585,430 180x95), "%s", text variable: ref.config.knownPositions.position19.name, invisible if: widget.invisiblePosition19, input disabled if: ref.processes.moveKnownPosition.statuses.enabledStatus.disabled
        OnMouseClick: execute { ref.processes.moveKnownPosition.request(ref.config.knownPositions.position19.name); }
END_VISUALIZATION

// ---- MTCS/Axes/Visu/VISU_AxesManual_MoveAbsolute.TcVIS
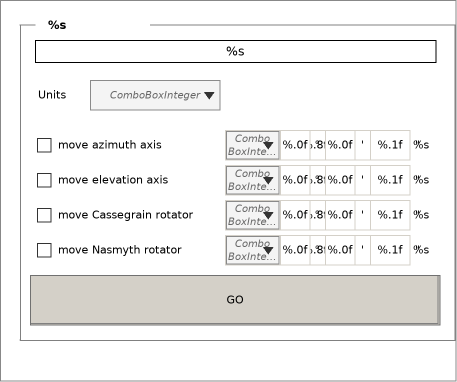
VISUALIZATION VISU_AxesManual_MoveAbsolute  // 457x382
VAR_IN_OUT
	ref : Axes;
    widget : AxesManualMoveAbsoluteWidget;
END_VAR
    Frame (15,10 440x370)
        shows VISU_AxesMultiMoveProcess(ref := ref.processes.moveAbsolute, widget := widget.moveAbsolute)
END_VISUALIZATION

// ---- MTCS/Axes/Visu/VISU_Axes_Commands_Power.TcVIS
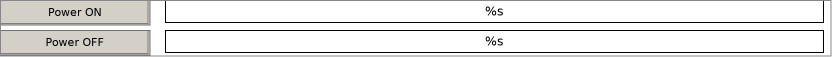
VISUALIZATION VISU_Axes_Commands_Power  // 832x57
VAR_IN_OUT
	powerOn : AxesPowerOnProcess;
    powerOff : AxesPowerOffProcess;
    
    powerOnStatus : StatusWidget;
    powerOffStatus : StatusWidget;
    
END_VAR
    Button (0,0 150x25), "Power ON", input disabled if: powerOn.statuses.enabledStatus.disabled
        OnMouseClick: execute { powerOn.request(); }
    Button (0,30 150x25), "Power OFF", input disabled if: powerOff.statuses.enabledStatus.disabled
        OnMouseClick: execute { powerOff.request(); }
    Frame (165,0 665x25)
        shows VISU_StatusWidget(widget := powerOnStatus)
    Frame (165,30 665x25)
        shows VISU_StatusWidget(widget := powerOffStatus)
END_VISUALIZATION

// ---- MTCS/Axes/Visu/VISU_AxesElevationAxis_Overview.TcVIS
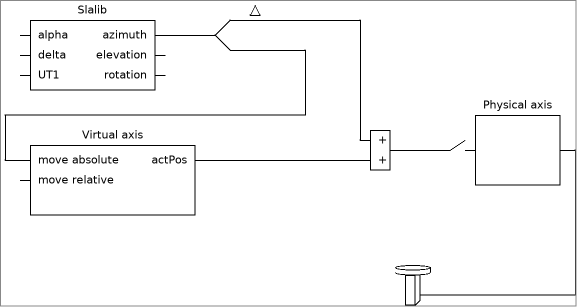
VISUALIZATION VISU_AxesElevationAxis_Overview  // 577x307
VAR_IN_OUT
	ref : AxesElevationAxis;
    widget : AxesElevationAxisWidget;
END_VAR
    Rectangle (405,275 10x30)
    Rectangle (30,20 125x70)
    Line (20,35) (30,35)
    Label (35,25 50x20), "alpha"
    Line (20,55) (30,55)
    Label (35,45 50x20), "delta"
    Line (20,75) (30,75)
    Label (35,65 50x20), "UT1"
    Polyline (255,5) (250,15) (260,15) (255,5)
    Label (30,0 125x20), "Slalib"
    Label (95,25 55x20), "azimuth"
    Label (90,45 60x20), "elevation"
    Label (100,65 50x20), "rotation"
    Line (155,55) (165,55)
    Line (155,75) (165,75)
    Rectangle (30,145 165x70)
    Label (35,150 95x20), "move absolute"
    Line (20,180) (30,180)
    Label (35,170 85x20), "move relative"
    Label (30,125 165x20), "Virtual axis"
    Label (135,150 55x20), "actPos"
    Polyline (155,35) (215,35) (230,50)
    Polyline (230,50) (305,50) (305,115) (5,115) (5,160) (30,160)
    Polyline (215,35) (230,20) (360,20) (360,140) (370,140)
    Polyline (195,160) (370,160)
    Rectangle (370,130 20x40)
    Label (375,130 15x20), "+"
    Label (375,150 15x20), "+"
    Line (390,150) (450,150)
    Line (450,150) (465,140)
    Line (465,150) (475,150)
    Rectangle (475,115 85x70)
    Label (475,95 85x20), "Physical axis"
    Polyline (560,150) (575,150) (575,295) (420,295)
    Polyline (415,305) (420,300) (420,275)
    Ellipse (395,270 35x5)
    Rectangle (395,270 35x2)
    Ellipse (395,265 35x5)
    Line (430,267) (430,272)
END_VISUALIZATION

// ---- MTCS/Axes/Visu/VISU_AxesElevationAxis_AbsoluteEncoder.TcVIS
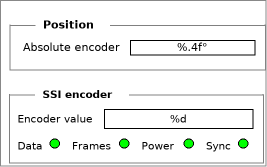
VISUALIZATION VISU_AxesElevationAxis_AbsoluteEncoder  // 267x167
VAR_IN_OUT
	ref : AxesElevationAxis;
    widget : AxesElevationAxisWidget;
END_VAR
    Frame (-5,80 270x85)
        shows VISU_SSIEncoder(ref := ref.parts.absoluteEncoder)
    Label (40,15 65x20), "Position"
    Polyline (110,25) (265,25) (265,70) (10,70) (10,25) (35,25)
    Label (20,40 105x15), "Absolute encoder"
    Rectangle (130,40 125x15), "%.4f°", text variable: ref.absoluteEncoderPosition.degrees.value
END_VISUALIZATION

// ---- MTCS/Axes/Visu/VISU_AxesElevationAxis_Lidas.TcVIS
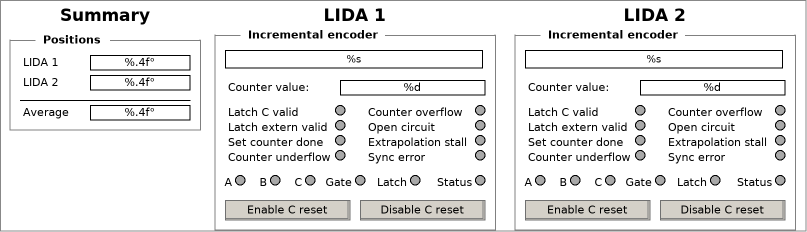
VISUALIZATION VISU_AxesElevationAxis_Lidas  // 807x232
VAR_IN_OUT
	ref : AxesElevationAxis;
    widget : AxesElevationAxisWidget;
END_VAR
    Label (215,0 280x30), "LIDA 1"
    Frame (215,25 290x205)
        shows VISU_IncrementalEncoder(ref := ref.parts.lida1, widget := widget.lida1)
    Label (515,0 280x30), "LIDA 2"
    Frame (515,25 290x205)
        shows VISU_IncrementalEncoder(ref := ref.parts.lida2, widget := widget.lida2)
    Label (10,0 190x30), "Summary"
    Label (40,30 65x20), "Positions"
    Polyline (110,40) (200,40) (200,130) (10,130) (10,40) (35,40)
    Label (20,55 90x15), "LIDA 1"
    Rectangle (90,55 100x15), "%.4f°", text variable: ref.lida1Position.degrees.value
    Rectangle (90,75 100x15), "%.4f°", text variable: ref.lida2Position.degrees.value
    Label (20,75 90x15), "LIDA 2"
    Label (20,105 90x15), "Average"
    Rectangle (90,105 100x15), "%.4f°", text variable: ref.lidaAveragePosition.degrees.value
    Line (20,100) (190,100)
END_VISUALIZATION

// ---- MTCS/Axes/Visu/VISU_AxesAzimuthAxis_Overview.TcVIS
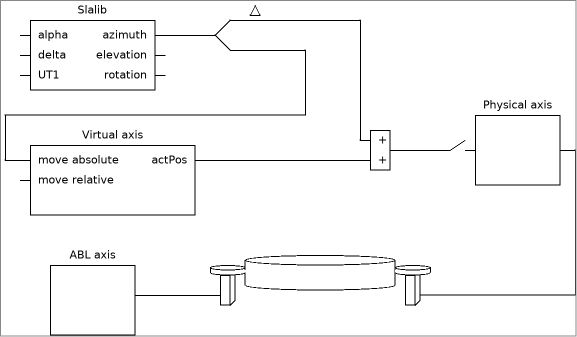
VISUALIZATION VISU_AxesAzimuthAxis_Overview  // 577x337
VAR_IN_OUT
	ref : AxesAzimuthAxis;
    widget : AxesAzimuthAxisWidget;
END_VAR
    Rectangle (405,275 10x30)
    Rectangle (30,20 125x70)
    Line (20,35) (30,35)
    Label (35,25 50x20), "alpha"
    Line (20,55) (30,55)
    Label (35,45 50x20), "delta"
    Line (20,75) (30,75)
    Label (35,65 50x20), "UT1"
    Polyline (255,5) (250,15) (260,15) (255,5)
    Label (30,0 125x20), "Slalib"
    Label (95,25 55x20), "azimuth"
    Label (90,45 60x20), "elevation"
    Label (100,65 50x20), "rotation"
    Line (155,55) (165,55)
    Line (155,75) (165,75)
    Rectangle (30,145 165x70)
    Label (35,150 95x20), "move absolute"
    Line (20,180) (30,180)
    Label (35,170 85x20), "move relative"
    Label (30,125 165x20), "Virtual axis"
    Label (135,150 55x20), "actPos"
    Polyline (155,35) (215,35) (230,50)
    Polyline (230,50) (305,50) (305,115) (5,115) (5,160) (30,160)
    Polyline (215,35) (230,20) (360,20) (360,140) (370,140)
    Polyline (195,160) (370,160)
    Rectangle (370,130 20x40)
    Label (375,130 15x20), "+"
    Label (375,150 15x20), "+"
    Line (390,150) (450,150)
    Line (450,150) (465,140)
    Line (465,150) (475,150)
    Rectangle (475,115 85x70)
    Label (475,95 85x20), "Physical axis"
    Polyline (560,150) (575,150) (575,295) (420,295)
    Rectangle (50,265 85x70)
    Label (50,245 85x20), "ABL axis"
    Ellipse (245,280 150x10)
    Rectangle (245,260 150x25)
    Ellipse (245,255 150x10)
    Line (245,285) (245,260)
    Line (395,285) (395,260)
    Polyline (415,305) (420,300) (420,275)
    Ellipse (395,270 35x5)
    Rectangle (395,270 35x2)
    Ellipse (395,265 35x5)
    Line (430,267) (430,272)
    Rectangle (220,275 10x30)
    Polyline (230,305) (235,300) (235,275)
    Ellipse (210,270 35x5)
    Rectangle (210,270 35x2)
    Ellipse (210,265 35x5)
    Line (210,267) (210,272)
    Polyline (135,295) (220,295)
END_VISUALIZATION

// ---- MTCS/Axes/Visu/VISU_AxesAzimuthAxis_Lidas.TcVIS
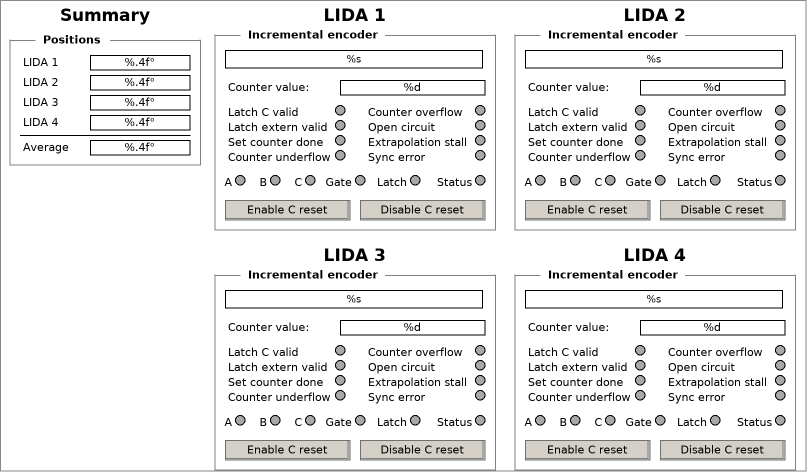
VISUALIZATION VISU_AxesAzimuthAxis_Lidas  // 807x472
VAR_IN_OUT
	ref : AxesAzimuthAxis;
    widget : AxesAzimuthAxisWidget;
END_VAR
    Label (215,0 280x30), "LIDA 1"
    Frame (215,25 290x205)
        shows VISU_IncrementalEncoder(ref := ref.parts.lida1, widget := widget.lida1)
    Label (215,240 280x30), "LIDA 3"
    Frame (215,265 290x205)
        shows VISU_IncrementalEncoder(ref := ref.parts.lida3, widget := widget.lida3)
    Label (515,0 280x30), "LIDA 2"
    Frame (515,25 290x205)
        shows VISU_IncrementalEncoder(ref := ref.parts.lida2, widget := widget.lida2)
    Label (515,240 280x30), "LIDA 4"
    Frame (515,265 290x205)
        shows VISU_IncrementalEncoder(ref := ref.parts.lida4, widget := widget.lida4)
    Label (10,0 190x30), "Summary"
    Label (40,30 65x20), "Positions"
    Polyline (110,40) (200,40) (200,165) (10,165) (10,40) (35,40)
    Label (20,55 90x15), "LIDA 1"
    Rectangle (90,55 100x15), "%.4f°", text variable: ref.lida1Position.degrees.value
    Rectangle (90,75 100x15), "%.4f°", text variable: ref.lida2Position.degrees.value
    Label (20,75 90x15), "LIDA 2"
    Rectangle (90,95 100x15), "%.4f°", text variable: ref.lida3Position.degrees.value
    Label (20,95 90x15), "LIDA 3"
    Rectangle (90,115 100x15), "%.4f°", text variable: ref.lida4Position.degrees.value
    Label (20,115 90x15), "LIDA 4"
    Label (20,140 90x15), "Average"
    Rectangle (90,140 100x15), "%.4f°", text variable: ref.lidaAveragePosition.degrees.value
    Line (20,135) (190,135)
END_VISUALIZATION

// ---- MTCS/Axes/Visu/VISU_AxesConfig_Azimuth_1.TcVIS
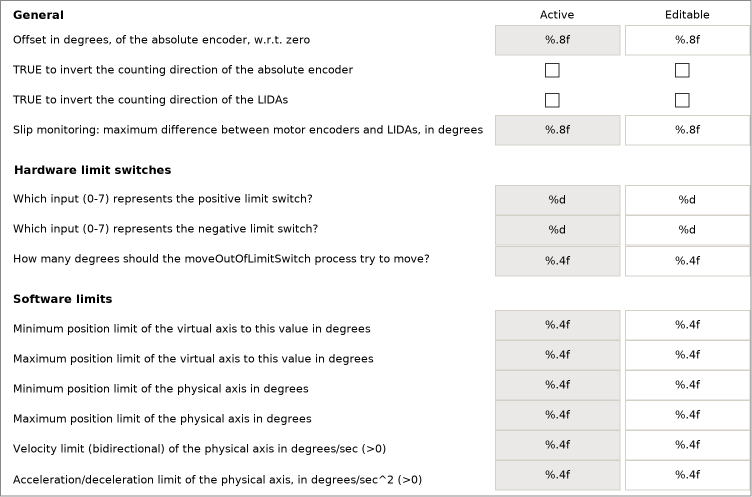
VISUALIZATION VISU_AxesConfig_Azimuth_1  // 752x497
VAR_IN_OUT
    active : AxesAzimuthConfig;
    editable : AxesAzimuthConfig;
END_VAR
    Label (495,5 125x20), "Active"
    Label (625,5 125x20), "Editable"
    Label (10,25 360x30), "Offset in degrees, of the absolute encoder, w.r.t. zero"
    Frame (495,25 255x30)
        shows VISU_ConfigLREAL8Entry(active := active.absoluteEncoderOffset, editable := editable.absoluteEncoderOffset)
    Label (10,184 475x30), "Which input (0-7) represents the positive limit switch?"
    Label (10,214 475x30), "Which input (0-7) represents the negative limit switch?"
    Label (10,244 475x30), "How many degrees should the moveOutOfLimitSwitch process try to move?"
    Label (11,155 150x30), "Hardware limit switches"
    Label (10,314 475x30), "Minimum position limit of the virtual axis to this value in degrees"
    Label (10,284 165x30), "Software limits"
    Label (10,344 475x30), "Maximum position limit of the virtual axis to this value in degrees"
    Label (10,374 475x30), "Minimum position limit of the physical axis in degrees"
    Label (10,404 475x30), "Maximum position limit of the physical axis in degrees"
    Label (10,434 475x30), "Velocity limit (bidirectional) of the physical axis in degrees/sec (>0)"
    Label (10,465 475x30), "Acceleration/deceleration limit of the physical axis, in degrees/sec^2 (>0)"
    Label (10,115 480x30), "Slip monitoring: maximum difference between motor encoders and LIDAs, in degrees"
    Label (10,0 150x30), "General"
    Frame (495,185 255x30)
        shows VISU_ConfigSINTEntry(active := active.positiveLimitSwitchInput, editable := editable.positiveLimitSwitchInput)
    Frame (495,215 255x30)
        shows VISU_ConfigSINTEntry(active := active.negativeLimitSwitchInput, editable := editable.negativeLimitSwitchInput)
    Frame (495,246 255x30)
        shows VISU_ConfigLREAL4Entry(active := active.moveOutOfLimitSwitchDistance, editable := editable.moveOutOfLimitSwitchDistance)
    Frame (495,310 255x30)
        shows VISU_ConfigLREAL4Entry(active := active.minPositionLimitVirtualAxis, editable := editable.minPositionLimitVirtualAxis)
    Frame (495,340 255x30)
        shows VISU_ConfigLREAL4Entry(active := active.maxPositionLimitVirtualAxis, editable := editable.maxPositionLimitVirtualAxis)
    Frame (495,370 255x30)
        shows VISU_ConfigLREAL4Entry(active := active.minPositionLimitPhysicalAxis, editable := editable.minPositionLimitPhysicalAxis)
    Frame (495,400 255x30)
        shows VISU_ConfigLREAL4Entry(active := active.maxPositionLimitPhysicalAxis, editable := editable.maxPositionLimitPhysicalAxis)
    Frame (495,430 255x30)
        shows VISU_ConfigLREAL4Entry(active := active.velocityLimit, editable := editable.velocityLimit)
    Frame (495,460 255x30)
        shows VISU_ConfigLREAL4Entry(active := active.accelerationLimit, editable := editable.accelerationLimit)
    Frame (495,55 255x30)
        shows VISU_ConfigBOOLEntry(active := active.absoluteEncoderInvert, editable := editable.absoluteEncoderInvert)
    Frame (495,115 255x30)
        shows VISU_ConfigLREAL8Entry(active := active.slipLimit, editable := editable.slipLimit)
    Label (10,55 360x30), "TRUE to invert the counting direction of the absolute encoder"
    Frame (495,85 255x30)
        shows VISU_ConfigBOOLEntry(active := active.lidasInvert, editable := editable.lidasInvert)
    Label (10,85 360x30), "TRUE to invert the counting direction of the LIDAs"
END_VISUALIZATION

// ---- MTCS/Axes/Visu/VISU_AxesConfig_Azimuth_3.TcVIS
